LIN {X 0,Y 255.969,Z 835.136,A -85,B 0,C 180,E1 -27165.742,E2 -27165.742} C_VEL
LIN {X 0,Y 253.083,Z 837.367,A -85,B 0,C 180,E1 -27167.208,E2 -27167.208} C_VEL
LIN {X 0,Y 247.96,Z 840.393,A -85,B 0,C 180,E1 -27170.241,E2 -27170.241} C_VEL
LIN {X 0,Y 243.682,Z 841.765,A -85,B 0,C 180,E1 -27173.397,E2 -27173.397} C_VEL
LIN {X 0,Y 241.91,Z 841.979,A -85,B 0,C 180,E1 -27175.016,E2 -27175.016} C_VEL
LIN {X 0,Y 239.218,Z 841.037,A -85,B 0,C 180,E1 -27178.322,E2 -27178.322} C_VEL
LIN {X 0,Y 237.369,Z 838.544,A -85,B 0,C 180,E1 -27181.69,E2 -27181.69} C_VEL
LIN {X 0,Y 236.528,Z 835.644,A -85,B 0,C 180,E1 -27184.245,E2 -27184.245} C_VEL
LIN {X 0,Y 236.07,Z 831.744,A -85,B 0,C 180,E1 -27186.816,E2 -27186.816} C_VEL
LIN {X 0,Y 236.118,Z 826.783,A -85,B 0,C 180,E1 -27189.39,E2 -27189.39} C_VEL
LIN {X 0,Y 236.294,Z 821.698,A -85,B 0,C 180,E1 -27191.551,E2 -27191.551} C_VEL
LIN {X 0,Y 236.654,Z 814.142,A -85,B 0,C 180,E1 -27194.133,E2 -27194.133} C_VEL
LIN {X 0,Y 237.029,Z 806.345,A -85,B 0,C 180,E1 -27196.303,E2 -27196.303} C_VEL
LIN {X 0,Y 237.449,Z 797.897,A -85,B 0,C 180,E1 -27198.265,E2 -27198.265} C_VEL
LIN {X 0,Y 237.963,Z 788.686,A -85,B 0,C 180,E1 -27200.055,E2 -27200.055} C_VEL
LIN {X 0,Y 238.5,Z 779.618,A -85,B 0,C 180,E1 -27201.537,E2 -27201.537} C_VEL
LIN {X 0,Y 239.065,Z 770.085,A -85,B 0,C 180,E1 -27202.843,E2 -27202.843} C_VEL
LIN {X 0,Y 239.688,Z 759.488,A -85,B 0,C 180,E1 -27204.034,E2 -27204.034} C_VEL
LIN {X 0,Y 240.123,Z 749.746,A -85,B 0,C 180,E1 -27204.918,E2 -27204.918} C_VEL
LIN {X 0,Y 240.469,Z 738.64,A -85,B 0,C 180,E1 -27205.698,E2 -27205.698} C_VEL
LIN {X 0,Y 241.686,Z 705.322,A -85,B 0,C 180,E1 -27207.392,E2 -27207.392} C_VEL
LIN {X 0,Y 242.808,Z 665.259,A -85,B 0,C 180,E1 -27209.316,E2 -27209.316} C_VEL
LIN {X 0,Y 240.288,Z 637.438,A -85,B 0,C 180,E1 -27210.679,E2 -27210.679} C_VEL
LIN {X 0,Y 239.995,Z 630.334,A -85,B 0,C 180,E1 -27211.063,E2 -27211.063} C_VEL
LIN {X 0,Y 239.543,Z 627.579,A -85,B 0,C 180,E1 -27212.273,E2 -27212.273} C_VEL
LIN {X 0,Y 239.08,Z 627.634,A -85,B 0,C 180,E1 -27217.969,E2 -27217.969} C_VEL
LIN {X 0,Y 239.069,Z 627.637,A -85,B 0,C 180,E1 -27222.366,E2 -27222.366} C_VEL
LIN {X 0,Y 239.081,Z 627.631,A -85,B 0,C 180,E1 -27225.32,E2 -27225.32} C_VEL
LIN {X 0,Y 239.062,Z 627.639,A -85,B 0,C 180,E1 -27229.864,E2 -27229.864} C_VEL
LIN {X 0,Y 239.028,Z 627.641,A -85,B 0,C 180,E1 -27234.12,E2 -27234.12} C_VEL
LIN {X 0,Y 239.074,Z 627.638,A -85,B 0,C 180,E1 -27238.172,E2 -27238.172} C_VEL
LIN {X 0,Y 239.121,Z 627.632,A -85,B 0,C 180,E1 -27242.051,E2 -27242.051} C_VEL
LIN {X 0,Y 239.152,Z 627.623,A -85,B 0,C 180,E1 -27245.792,E2 -27245.792} C_VEL
LIN {X 0,Y 239.202,Z 627.62,A -85,B 0,C 180,E1 -27249.558,E2 -27249.558} C_VEL
LIN {X 0,Y 239.321,Z 627.599,A -85,B 0,C 180,E1 -27254.978,E2 -27254.978} C_VEL
LIN {X 0,Y 239.388,Z 627.599,A -85,B 0,C 180,E1 -27259.888,E2 -27259.888} C_VEL
LIN {X 0,Y 239.662,Z 627.561,A -85,B 0,C 180,E1 -27263.554,E2 -27263.554} C_VEL
LIN {X 0,Y 239.728,Z 627.552,A -85,B 0,C 180,E1 -27266.65,E2 -27266.65} C_VEL
LIN {X 0,Y 239.869,Z 627.54,A -85,B 0,C 180,E1 -27270,E2 -27270} C_VEL
LIN {X 0,Y 239.728,Z 627.552,A -85,B 0,C 180,E1 -27273.35,E2 -27273.35} C_VEL
LIN {X 0,Y 239.62,Z 627.566,A -85,B 0,C 180,E1 -27276.714,E2 -27276.714} C_VEL
LIN {X 0,Y 239.355,Z 627.603,A -85,B 0,C 180,E1 -27281.82,E2 -27281.82} C_VEL
LIN {X 0,Y 239.296,Z 627.603,A -85,B 0,C 180,E1 -27285.274,E2 -27285.274} C_VEL
LIN {X 0,Y 239.191,Z 627.621,A -85,B 0,C 180,E1 -27290.573,E2 -27290.573} C_VEL
LIN {X 0,Y 239.135,Z 627.623,A -85,B 0,C 180,E1 -27294.77,E2 -27294.77} C_VEL
LIN {X 0,Y 239.118,Z 627.631,A -85,B 0,C 180,E1 -27298.506,E2 -27298.506} C_VEL
LIN {X 0,Y 239.094,Z 627.635,A -85,B 0,C 180,E1 -27301.836,E2 -27301.836} C_VEL
LIN {X 0,Y 239.124,Z 627.628,A -85,B 0,C 180,E1 -27305.862,E2 -27305.862} C_VEL
LIN {X 0,Y 239.097,Z 627.633,A -85,B 0,C 180,E1 -27310.389,E2 -27310.389} C_VEL
LIN {X 0,Y 239.09,Z 627.63,A -85,B 0,C 180,E1 -27314.677,E2 -27314.677} C_VEL
LIN {X 0,Y 239.091,Z 627.634,A -85,B 0,C 180,E1 -27317.639,E2 -27317.639} C_VEL
LIN {X 0,Y 239.091,Z 627.633,A -85,B 0,C 180,E1 -27322.033,E2 -27322.033} C_VEL
LIN {X 0,Y 239.093,Z 627.635,A -85,B 0,C 180,E1 -27326.178,E2 -27326.178} C_VEL
LIN {X 0,Y 239.071,Z 627.637,A -85,B 0,C 180,E1 -27330.128,E2 -27330.128} C_VEL
LIN {X 0,Y 239.107,Z 627.629,A -85,B 0,C 180,E1 -27333.934,E2 -27333.934} C_VEL
LIN {X 0,Y 239.112,Z 627.632,A -85,B 0,C 180,E1 -27337.616,E2 -27337.616} C_VEL
LIN {X 0,Y 239.174,Z 627.621,A -85,B 0,C 180,E1 -27341.208,E2 -27341.208} C_VEL
LIN {X 0,Y 239.271,Z 627.609,A -85,B 0,C 180,E1 -27345.026,E2 -27345.026} C_VEL
LIN {X 0,Y 239.384,Z 627.6,A -85,B 0,C 180,E1 -27349.889,E2 -27349.889} C_VEL
LIN {X 0,Y 239.717,Z 627.551,A -85,B 0,C 180,E1 -27353.446,E2 -27353.446} C_VEL
LIN {X 0,Y 239.736,Z 627.553,A -85,B 0,C 180,E1 -27356.651,E2 -27356.651} C_VEL
LIN {X 0,Y 239.87,Z 627.538,A -85,B 0,C 180,E1 -27360.001,E2 -27360.001} C_VEL
LIN {X 0,Y 239.73,Z 627.549,A -85,B 0,C 180,E1 -27363.351,E2 -27363.351} C_VEL
LIN {X 0,Y 239.623,Z 627.567,A -85,B 0,C 180,E1 -27366.715,E2 -27366.715} C_VEL
LIN {X 0,Y 239.305,Z 627.605,A -85,B 0,C 180,E1 -27371.823,E2 -27371.823} C_VEL
LIN {X 0,Y 239.217,Z 627.617,A -85,B 0,C 180,E1 -27375.28,E2 -27375.28} C_VEL
LIN {X 0,Y 239.138,Z 627.624,A -85,B 0,C 180,E1 -27380.579,E2 -27380.579} C_VEL
LIN {X 0,Y 239.138,Z 627.627,A -85,B 0,C 180,E1 -27384.77,E2 -27384.77} C_VEL
LIN {X 0,Y 239.118,Z 627.63,A -85,B 0,C 180,E1 -27388.504,E2 -27388.504} C_VEL
LIN {X 0,Y 239.076,Z 627.633,A -85,B 0,C 180,E1 -27391.828,E2 -27391.828} C_VEL
LIN {X 0,Y 239.028,Z 627.644,A -85,B 0,C 180,E1 -27395.88,E2 -27395.88} C_VEL
LIN {X 0,Y 239.059,Z 627.635,A -85,B 0,C 180,E1 -27400.136,E2 -27400.136} C_VEL
LIN {X 0,Y 239.041,Z 627.64,A -85,B 0,C 180,E1 -27404.689,E2 -27404.689} C_VEL
LIN {X 0,Y 239.021,Z 627.643,A -85,B 0,C 180,E1 -27407.623,E2 -27407.623} C_VEL
LIN {X 0,Y 239.055,Z 627.636,A -85,B 0,C 180,E1 -27412.026,E2 -27412.026} C_VEL
LIN {X 0,Y 239.072,Z 627.638,A -85,B 0,C 180,E1 -27416.174,E2 -27416.174} C_VEL
LIN {X 0,Y 239.09,Z 627.631,A -85,B 0,C 180,E1 -27420.13,E2 -27420.13} C_VEL
LIN {X 0,Y 239.45,Z 627.719,A -85,B 0,C 180,E1 -27423.565,E2 -27423.565} C_VEL
LIN {X 0,Y 240.611,Z 633.644,A -85,B 0,C 180,E1 -27425.949,E2 -27425.949} C_VEL
LIN {X 0,Y 240.293,Z 637.031,A -85,B 0,C 180,E1 -27427.28,E2 -27427.28} C_VEL
LIN {X 0,Y 239.534,Z 641.423,A -85,B 0,C 180,E1 -27428.963,E2 -27428.963} C_VEL
LIN {X 0,Y 240.199,Z 661.866,A -85,B 0,C 180,E1 -27429.962,E2 -27429.962} C_VEL
LIN {X 0,Y 242.502,Z 689.559,A -85,B 0,C 180,E1 -27431.311,E2 -27431.311} C_VEL
LIN {X 0,Y 240.805,Z 746.631,A -85,B 0,C 180,E1 -27434.117,E2 -27434.117} C_VEL
LIN {X 0,Y 240.33,Z 758.435,A -85,B 0,C 180,E1 -27434.901,E2 -27434.901} C_VEL
LIN {X 0,Y 239.916,Z 769.202,A -85,B 0,C 180,E1 -27435.847,E2 -27435.847} C_VEL
LIN {X 0,Y 239.736,Z 772.319,A -85,B 0,C 180,E1 -27436.16,E2 -27436.16} C_VEL
LIN {X 0,Y 239.264,Z 775.883,A -85,B 0,C 180,E1 -27436.545,E2 -27436.545} C_VEL
LIN {X 0,Y 236.945,Z 782.54,A -85,B 0,C 180,E1 -27437.412,E2 -27437.412} C_VEL
LIN {X 0,Y 232.121,Z 793.434,A -85,B 0,C 180,E1 -27439.214,E2 -27439.214} C_VEL
LIN {X 0,Y 231.246,Z 798.101,A -85,B 0,C 180,E1 -27440.079,E2 -27440.079} C_VEL
LIN {X 0,Y 230.873,Z 806.382,A -85,B 0,C 180,E1 -27441.715,E2 -27441.715} C_VEL
LIN {X 0,Y 230.528,Z 813.892,A -85,B 0,C 180,E1 -27443.458,E2 -27443.458} C_VEL
LIN {X 0,Y 230.407,Z 820.396,A -85,B 0,C 180,E1 -27445.205,E2 -27445.205} C_VEL
LIN {X 0,Y 230.245,Z 827.124,A -85,B 0,C 180,E1 -27447.385,E2 -27447.385} C_VEL
LIN {X 0,Y 230.066,Z 833.651,A -85,B 0,C 180,E1 -27450,E2 -27450} C_VEL
LIN {X 0,Y 229.927,Z 837.306,A -85,B 0,C 180,E1 -27451.746,E2 -27451.746} C_VEL
LIN {X 0,Y 229.564,Z 842.85,A -85,B 0,C 180,E1 -27455.252,E2 -27455.252} C_VEL
LIN {X 0,Y 229.53,Z 844.969,A -85,B 0,C 180,E1 -27457.012,E2 -27457.012} C_VEL
LIN {X 0,Y 230.453,Z 848.056,A -85,B 0,C 180,E1 -27460.508,E2 -27460.508} C_VEL
LIN {X 0,Y 232.38,Z 849.575,A -85,B 0,C 180,E1 -27463.954,E2 -27463.954} C_VEL
LIN {X 0,Y 235.467,Z 849.632,A -85,B 0,C 180,E1 -27467.306,E2 -27467.306} C_VEL
LIN {X 0,Y 237.383,Z 849.211,A -85,B 0,C 180,E1 -27468.94,E2 -27468.94} C_VEL
LIN {X 0,Y 241.904,Z 847.088,A -85,B 0,C 180,E1 -27472.113,E2 -27472.113} C_VEL
LIN {X 0,Y 245.879,Z 844.5,A -85,B 0,C 180,E1 -27474.398,E2 -27474.398} C_VEL
LIN {X 0,Y 252.044,Z 839.532,A -85,B 0,C 180,E1 -27477.294,E2 -27477.294} C_VEL
LIN {X 0,Y 257.146,Z 834.695,A -85,B 0,C 180,E1 -27479.361,E2 -27479.361} C_VEL
LIN {X 0,Y 262.686,Z 828.671,A -85,B 0,C 180,E1 -27481.33,E2 -27481.33} C_VEL
LIN {X 0,Y 268.677,Z 821.348,A -85,B 0,C 180,E1 -27483.194,E2 -27483.194} C_VEL
LIN {X 0,Y 273.992,Z 814.098,A -85,B 0,C 180,E1 -27484.668,E2 -27484.668} C_VEL
LIN {X 0,Y 279.55,Z 805.482,A -85,B 0,C 180,E1 -27486.074,E2 -27486.074} C_VEL
LIN {X 0,Y 284.285,Z 797.291,A -85,B 0,C 180,E1 -27487.132,E2 -27487.132} C_VEL
LIN {X 0,Y 289.766,Z 786.418,A -85,B 0,C 180,E1 -27488.275,E2 -27488.275} C_VEL
LIN {X 0,Y 294.221,Z 776.249,A -85,B 0,C 180,E1 -27489.115,E2 -27489.115} C_VEL
LIN {X 0,Y 298.033,Z 765.844,A -85,B 0,C 180,E1 -27489.825,E2 -27489.825} C_VEL
LIN {X 0,Y 301.383,Z 754.97,A -85,B 0,C 180,E1 -27490.38,E2 -27490.38} C_VEL
LIN {X 0,Y 304.7,Z 740.723,A -85,B 0,C 180,E1 -27490.982,E2 -27490.982} C_VEL
LIN {X 0,Y 306.247,Z 732.083,A -85,B 0,C 180,E1 -27491.312,E2 -27491.312} C_VEL
LIN {X 0,Y 304.844,Z 726.881,A -85,B 0,C 180,E1 -27493.21,E2 -27493.21} C_VEL
LIN {X 0,Y 303.582,Z 722.992,A -85,B 0,C 180,E1 -27495.274,E2 -27495.274} C_VEL
LIN {X 0,Y 302.655,Z 719.169,A -85,B 0,C 180,E1 -27498.363,E2 -27498.363} C_VEL
LIN {X 0,Y 302.452,Z 718.617,A -85,B 0,C 180,E1 -27499.84,E2 -27499.84} C_VEL
LIN {X 0,Y 302.826,Z 718.852,A -85,B 0,C 180,E1 -27502.516,E2 -27502.516} C_VEL
LIN {X 0,Y 304.244,Z 722.091,A -85,B 0,C 180,E1 -27505.819,E2 -27505.819} C_VEL
LIN {X 0,Y 305.607,Z 725.321,A -85,B 0,C 180,E1 -27507.638,E2 -27507.638} C_VEL
LIN {X 0,Y 306.67,Z 728.479,A -85,B 0,C 180,E1 -27508.958,E2 -27508.958} C_VEL
LIN {X 0,Y 302.997,Z 746.766,A -85,B 0,C 180,E1 -27509.657,E2 -27509.657} C_VEL
LIN {X 0,Y 299.281,Z 759.828,A -85,B 0,C 180,E1 -27510.346,E2 -27510.346} C_VEL
LIN {X 0,Y 295.517,Z 770.423,A -85,B 0,C 180,E1 -27511.064,E2 -27511.064} C_VEL
LIN {X 0,Y 291.043,Z 781.07,A -85,B 0,C 180,E1 -27512.011,E2 -27512.011} C_VEL
LIN {X 0,Y 286.235,Z 790.813,A -85,B 0,C 180,E1 -27513.082,E2 -27513.082} C_VEL
LIN {X 0,Y 282.131,Z 798.294,A -85,B 0,C 180,E1 -27514.071,E2 -27514.071} C_VEL
LIN {X 0,Y 277.047,Z 806.464,A -85,B 0,C 180,E1 -27515.39,E2 -27515.39} C_VEL
LIN {X 0,Y 271.848,Z 813.824,A -85,B 0,C 180,E1 -27516.863,E2 -27516.863} C_VEL
LIN {X 0,Y 266.753,Z 820.185,A -85,B 0,C 180,E1 -27518.431,E2 -27518.431} C_VEL
LIN {X 0,Y 261.584,Z 825.975,A -85,B 0,C 180,E1 -27520.187,E2 -27520.187} C_VEL
LIN {X 0,Y 257.596,Z 830.02,A -85,B 0,C 180,E1 -27521.695,E2 -27521.695} C_VEL
LIN {X 0,Y 252.276,Z 834.546,A -85,B 0,C 180,E1 -27523.88,E2 -27523.88} C_VEL
LIN {X 0,Y 246.147,Z 838.668,A -85,B 0,C 180,E1 -27526.841,E2 -27526.841} C_VEL
LIN {X 0,Y 242.87,Z 840.464,A -85,B 0,C 180,E1 -27528.689,E2 -27528.689} C_VEL
LIN {X 0,Y 238.623,Z 841.904,A -85,B 0,C 180,E1 -27531.56,E2 -27531.56} C_VEL
LIN {X 0,Y 234.798,Z 842.001,A -85,B 0,C 180,E1 -27534.865,E2 -27534.865} C_VEL
LIN {X 0,Y 233.286,Z 841.573,A -85,B 0,C 180,E1 -27536.557,E2 -27536.557} C_VEL
LIN {X 0,Y 231.064,Z 839.415,A -85,B 0,C 180,E1 -27539.999,E2 -27539.999} C_VEL
LIN {X 0,Y 229.918,Z 836.807,A -85,B 0,C 180,E1 -27542.619,E2 -27542.619} C_VEL
LIN {X 0,Y 229.245,Z 833.24,A -85,B 0,C 180,E1 -27545.259,E2 -27545.259} C_VEL
LIN {X 0,Y 229.024,Z 828.587,A -85,B 0,C 180,E1 -27547.91,E2 -27547.91} C_VEL
LIN {X 0,Y 229.285,Z 821.172,A -85,B 0,C 180,E1 -27551.175,E2 -27551.175} C_VEL
LIN {X 0,Y 229.589,Z 814.033,A -85,B 0,C 180,E1 -27553.676,E2 -27553.676} C_VEL
LIN {X 0,Y 229.903,Z 808.052,A -85,B 0,C 180,E1 -27555.46,E2 -27555.46} C_VEL
LIN {X 0,Y 230.325,Z 798.974,A -85,B 0,C 180,E1 -27557.704,E2 -27557.704} C_VEL
LIN {X 0,Y 230.833,Z 790.228,A -85,B 0,C 180,E1 -27559.498,E2 -27559.498} C_VEL
LIN {X 0,Y 231.31,Z 781.035,A -85,B 0,C 180,E1 -27561.083,E2 -27561.083} C_VEL
LIN {X 0,Y 231.965,Z 770.074,A -85,B 0,C 180,E1 -27562.643,E2 -27562.643} C_VEL
LIN {X 0,Y 232.541,Z 760.56,A -85,B 0,C 180,E1 -27563.757,E2 -27563.757} C_VEL
LIN {X 0,Y 233.025,Z 749.841,A -85,B 0,C 180,E1 -27564.767,E2 -27564.767} C_VEL
LIN {X 0,Y 233.376,Z 739.04,A -85,B 0,C 180,E1 -27565.553,E2 -27565.553} C_VEL
LIN {X 0,Y 234.237,Z 715.097,A -85,B 0,C 180,E1 -27566.83,E2 -27566.83} C_VEL
LIN {X 0,Y 235.787,Z 666.248,A -85,B 0,C 180,E1 -27569.3,E2 -27569.3} C_VEL
LIN {X 0,Y 233.191,Z 637.147,A -85,B 0,C 180,E1 -27570.768,E2 -27570.768} C_VEL
LIN {X 0,Y 232.898,Z 630.557,A -85,B 0,C 180,E1 -27571.125,E2 -27571.125} C_VEL
LIN {X 0,Y 232.529,Z 628.453,A -85,B 0,C 180,E1 -27572.132,E2 -27572.132} C_VEL
LIN {X 0,Y 232.013,Z 628.516,A -85,B 0,C 180,E1 -27578.285,E2 -27578.285} C_VEL
LIN {X 0,Y 232.009,Z 628.517,A -85,B 0,C 180,E1 -27581.619,E2 -27581.619} C_VEL
LIN {X 0,Y 232.034,Z 628.51,A -85,B 0,C 180,E1 -27586.028,E2 -27586.028} C_VEL
LIN {X 0,Y 231.995,Z 628.518,A -85,B 0,C 180,E1 -27590.651,E2 -27590.651} C_VEL
LIN {X 0,Y 232.012,Z 628.511,A -85,B 0,C 180,E1 -27594.997,E2 -27594.997} C_VEL
LIN {X 0,Y 232.016,Z 628.514,A -85,B 0,C 180,E1 -27599.121,E2 -27599.121} C_VEL
LIN {X 0,Y 232.062,Z 628.508,A -85,B 0,C 180,E1 -27603.079,E2 -27603.079} C_VEL
LIN {X 0,Y 232.082,Z 628.503,A -85,B 0,C 180,E1 -27606.899,E2 -27606.899} C_VEL
LIN {X 0,Y 232.135,Z 628.5,A -85,B 0,C 180,E1 -27610.615,E2 -27610.615} C_VEL
LIN {X 0,Y 232.283,Z 628.479,A -85,B 0,C 180,E1 -27616.04,E2 -27616.04} C_VEL
LIN {X 0,Y 232.402,Z 628.467,A -85,B 0,C 180,E1 -27621.332,E2 -27621.332} C_VEL
LIN {X 0,Y 232.593,Z 628.437,A -85,B 0,C 180,E1 -27624.816,E2 -27624.816} C_VEL
LIN {X 0,Y 232.694,Z 628.432,A -85,B 0,C 180,E1 -27628.275,E2 -27628.275} C_VEL
LIN {X 0,Y 232.835,Z 628.417,A -85,B 0,C 180,E1 -27630,E2 -27630} C_VEL
LIN {X 0,Y 232.696,Z 628.428,A -85,B 0,C 180,E1 -27633.451,E2 -27633.451} C_VEL
LIN {X 0,Y 232.545,Z 628.447,A -85,B 0,C 180,E1 -27636.92,E2 -27636.92} C_VEL
LIN {X 0,Y 232.289,Z 628.481,A -85,B 0,C 180,E1 -27642.185,E2 -27642.185} C_VEL
LIN {X 0,Y 232.199,Z 628.489,A -85,B 0,C 180,E1 -27645.753,E2 -27645.753} C_VEL
LIN {X 0,Y 232.155,Z 628.497,A -85,B 0,C 180,E1 -27650.723,E2 -27650.723} C_VEL
LIN {X 0,Y 232.085,Z 628.501,A -85,B 0,C 180,E1 -27655.123,E2 -27655.123} C_VEL
LIN {X 0,Y 232.057,Z 628.51,A -85,B 0,C 180,E1 -27658.916,E2 -27658.916} C_VEL
LIN {X 0,Y 232.051,Z 628.506,A -85,B 0,C 180,E1 -27662.91,E2 -27662.91} C_VEL
LIN {X 0,Y 232.051,Z 628.509,A -85,B 0,C 180,E1 -27667.135,E2 -27667.135} C_VEL
LIN {X 0,Y 232.029,Z 628.513,A -85,B 0,C 180,E1 -27671.615,E2 -27671.615} C_VEL
LIN {X 0,Y 232.041,Z 628.513,A -85,B 0,C 180,E1 -27676.031,E2 -27676.031} C_VEL
LIN {X 0,Y 232.031,Z 628.512,A -85,B 0,C 180,E1 -27680.66,E2 -27680.66} C_VEL
LIN {X 0,Y 232.055,Z 628.507,A -85,B 0,C 180,E1 -27685.006,E2 -27685.006} C_VEL
LIN {X 0,Y 232.016,Z 628.515,A -85,B 0,C 180,E1 -27689.122,E2 -27689.122} C_VEL
LIN {X 0,Y 232.063,Z 628.503,A -85,B 0,C 180,E1 -27693.08,E2 -27693.08} C_VEL
LIN {X 0,Y 232.072,Z 628.507,A -85,B 0,C 180,E1 -27696.899,E2 -27696.899} C_VEL
LIN {X 0,Y 232.114,Z 628.501,A -85,B 0,C 180,E1 -27700.614,E2 -27700.614} C_VEL
LIN {X 0,Y 232.228,Z 628.486,A -85,B 0,C 180,E1 -27704.835,E2 -27704.835} C_VEL
LIN {X 0,Y 232.308,Z 628.479,A -85,B 0,C 180,E1 -27709.578,E2 -27709.578} C_VEL
LIN {X 0,Y 232.666,Z 628.429,A -85,B 0,C 180,E1 -27713.447,E2 -27713.447} C_VEL
LIN {X 0,Y 232.705,Z 628.43,A -85,B 0,C 180,E1 -27716.549,E2 -27716.549} C_VEL
LIN {X 0,Y 232.835,Z 628.414,A -85,B 0,C 180,E1 -27720.001,E2 -27720.001} C_VEL
LIN {X 0,Y 232.699,Z 628.425,A -85,B 0,C 180,E1 -27723.452,E2 -27723.452} C_VEL
LIN {X 0,Y 232.548,Z 628.448,A -85,B 0,C 180,E1 -27726.92,E2 -27726.92} C_VEL
LIN {X 0,Y 232.235,Z 628.485,A -85,B 0,C 180,E1 -27732.189,E2 -27732.189} C_VEL
LIN {X 0,Y 232.153,Z 628.499,A -85,B 0,C 180,E1 -27735.757,E2 -27735.757} C_VEL
LIN {X 0,Y 232.084,Z 628.502,A -85,B 0,C 180,E1 -27740.675,E2 -27740.675} C_VEL
LIN {X 0,Y 232.088,Z 628.505,A -85,B 0,C 180,E1 -27745.123,E2 -27745.123} C_VEL
LIN {X 0,Y 232.056,Z 628.508,A -85,B 0,C 180,E1 -27748.915,E2 -27748.915} C_VEL
LIN {X 0,Y 232.01,Z 628.512,A -85,B 0,C 180,E1 -27752.918,E2 -27752.918} C_VEL
LIN {X 0,Y 231.995,Z 628.517,A -85,B 0,C 180,E1 -27757.146,E2 -27757.146} C_VEL
LIN {X 0,Y 231.978,Z 628.516,A -85,B 0,C 180,E1 -27761.627,E2 -27761.627} C_VEL
LIN {X 0,Y 231.972,Z 628.524,A -85,B 0,C 180,E1 -27766.014,E2 -27766.014} C_VEL
LIN {X 0,Y 231.993,Z 628.512,A -85,B 0,C 180,E1 -27770.651,E2 -27770.651} C_VEL
LIN {X 0,Y 232.012,Z 628.515,A -85,B 0,C 180,E1 -27774.998,E2 -27774.998} C_VEL
LIN {X 0,Y 232.025,Z 628.511,A -85,B 0,C 180,E1 -27779.123,E2 -27779.123} C_VEL
LIN {X 0,Y 232.431,Z 628.559,A -85,B 0,C 180,E1 -27783.722,E2 -27783.722} C_VEL
LIN {X 0,Y 233.539,Z 634.342,A -85,B 0,C 180,E1 -27786.115,E2 -27786.115} C_VEL
LIN {X 0,Y 232.455,Z 641.113,A -85,B 0,C 180,E1 -27788.858,E2 -27788.858} C_VEL
LIN {X 0,Y 233.082,Z 661.522,A -85,B 0,C 180,E1 -27789.904,E2 -27789.904} C_VEL
LIN {X 0,Y 235.356,Z 690.045,A -85,B 0,C 180,E1 -27791.342,E2 -27791.342} C_VEL
LIN {X 0,Y 233.731,Z 746.504,A -85,B 0,C 180,E1 -27794.246,E2 -27794.246} C_VEL
LIN {X 0,Y 233.288,Z 757.483,A -85,B 0,C 180,E1 -27794.992,E2 -27794.992} C_VEL
LIN {X 0,Y 232.885,Z 768.4,A -85,B 0,C 180,E1 -27795.967,E2 -27795.967} C_VEL
LIN {X 0,Y 232.378,Z 778.933,A -85,B 0,C 180,E1 -27797.156,E2 -27797.156} C_VEL
LIN {X 0,Y 231.772,Z 788.297,A -85,B 0,C 180,E1 -27798.451,E2 -27798.451} C_VEL
LIN {X 0,Y 231.362,Z 796.338,A -85,B 0,C 180,E1 -27799.755,E2 -27799.755} C_VEL
LIN {X 0,Y 231.246,Z 798.101,A -85,B 0,C 180,E1 -27800.079,E2 -27800.079} C_VEL
LIN {X 0,Y 230.404,Z 802.726,A -85,B 0,C 180,E1 -27800.965,E2 -27800.965} C_VEL
LIN {X 0,Y 227.31,Z 809.581,A -85,B 0,C 180,E1 -27802.589,E2 -27802.589} C_VEL
LIN {X 0,Y 224.235,Z 815.899,A -85,B 0,C 180,E1 -27804.391,E2 -27804.391} C_VEL
LIN {X 0,Y 223.469,Z 819.618,A -85,B 0,C 180,E1 -27805.566,E2 -27805.566} C_VEL
LIN {X 0,Y 223.313,Z 827.429,A -85,B 0,C 180,E1 -27808.203,E2 -27808.203} C_VEL
LIN {X 0,Y 223.147,Z 831.936,A -85,B 0,C 180,E1 -27810,E2 -27810} C_VEL
LIN {X 0,Y 222.817,Z 837.406,A -85,B 0,C 180,E1 -27812.703,E2 -27812.703} C_VEL
LIN {X 0,Y 222.587,Z 841.646,A -85,B 0,C 180,E1 -27815.417,E2 -27815.417} C_VEL
LIN {X 0,Y 222.854,Z 845.74,A -85,B 0,C 180,E1 -27819.042,E2 -27819.042} C_VEL
LIN {X 0,Y 224.423,Z 848.328,A -85,B 0,C 180,E1 -27822.62,E2 -27822.62} C_VEL
LIN {X 0,Y 225.504,Z 849.154,A -85,B 0,C 180,E1 -27824.389,E2 -27824.389} C_VEL
LIN {X 0,Y 228.697,Z 849.601,A -85,B 0,C 180,E1 -27827.835,E2 -27827.835} C_VEL
LIN {X 0,Y 233.413,Z 848.295,A -85,B 0,C 180,E1 -27831.522,E2 -27831.522} C_VEL
LIN {X 0,Y 238.017,Z 846.001,A -85,B 0,C 180,E1 -27834.331,E2 -27834.331} C_VEL
LIN {X 0,Y 242.556,Z 843.137,A -85,B 0,C 180,E1 -27836.59,E2 -27836.59} C_VEL
LIN {X 0,Y 247.543,Z 839.324,A -85,B 0,C 180,E1 -27838.753,E2 -27838.753} C_VEL
LIN {X 0,Y 252.95,Z 834.469,A -85,B 0,C 180,E1 -27840.816,E2 -27840.816} C_VEL
LIN {X 0,Y 259.515,Z 827.752,A -85,B 0,C 180,E1 -27842.993,E2 -27842.993} C_VEL
LIN {X 0,Y 265.128,Z 821.259,A -85,B 0,C 180,E1 -27844.612,E2 -27844.612} C_VEL
LIN {X 0,Y 270.652,Z 814.001,A -85,B 0,C 180,E1 -27846.07,E2 -27846.07} C_VEL
LIN {X 0,Y 276.447,Z 805.455,A -85,B 0,C 180,E1 -27847.452,E2 -27847.452} C_VEL
LIN {X 0,Y 281.999,Z 796.304,A -85,B 0,C 180,E1 -27848.614,E2 -27848.614} C_VEL
LIN {X 0,Y 286.434,Z 787.977,A -85,B 0,C 180,E1 -27849.48,E2 -27849.48} C_VEL
LIN {X 0,Y 290.998,Z 778.115,A -85,B 0,C 180,E1 -27850.308,E2 -27850.308} C_VEL
LIN {X 0,Y 294.944,Z 768.048,A -85,B 0,C 180,E1 -27851,E2 -27851} C_VEL
LIN {X 0,Y 298.418,Z 757.549,A -85,B 0,C 180,E1 -27851.566,E2 -27851.566} C_VEL
LIN {X 0,Y 301.567,Z 745.744,A -85,B 0,C 180,E1 -27852.078,E2 -27852.078} C_VEL
LIN {X 0,Y 303.56,Z 736.488,A -85,B 0,C 180,E1 -27852.415,E2 -27852.415} C_VEL
LIN {X 0,Y 302.477,Z 732.456,A -85,B 0,C 180,E1 -27854.056,E2 -27854.056} C_VEL
LIN {X 0,Y 301.739,Z 729.655,A -85,B 0,C 180,E1 -27855.586,E2 -27855.586} C_VEL
LIN {X 0,Y 300.957,Z 725.89,A -85,B 0,C 180,E1 -27858.725,E2 -27858.725} C_VEL
LIN {X 0,Y 300.891,Z 725.466,A -85,B 0,C 180,E1 -27861.058,E2 -27861.058} C_VEL
LIN {X 0,Y 301.183,Z 725.905,A -85,B 0,C 180,E1 -27862.621,E2 -27862.621} C_VEL
LIN {X 0,Y 302.366,Z 728.664,A -85,B 0,C 180,E1 -27865.454,E2 -27865.454} C_VEL
LIN {X 0,Y 303.657,Z 732.07,A -85,B 0,C 180,E1 -27867.388,E2 -27867.388} C_VEL
LIN {X 0,Y 303.935,Z 733.24,A -85,B 0,C 180,E1 -27867.828,E2 -27867.828} C_VEL
LIN {X 0,Y 300.28,Z 749.351,A -85,B 0,C 180,E1 -27868.471,E2 -27868.471} C_VEL
LIN {X 0,Y 296.74,Z 760.842,A -85,B 0,C 180,E1 -27869.09,E2 -27869.09} C_VEL
LIN {X 0,Y 292.661,Z 771.806,A -85,B 0,C 180,E1 -27869.827,E2 -27869.827} C_VEL
LIN {X 0,Y 288.946,Z 780.454,A -85,B 0,C 180,E1 -27870.58,E2 -27870.58} C_VEL
LIN {X 0,Y 284.491,Z 789.373,A -85,B 0,C 180,E1 -27871.508,E2 -27871.508} C_VEL
LIN {X 0,Y 279.02,Z 798.817,A -85,B 0,C 180,E1 -27872.732,E2 -27872.732} C_VEL
LIN {X 0,Y 273.188,Z 807.575,A -85,B 0,C 180,E1 -27874.159,E2 -27874.159} C_VEL
LIN {X 0,Y 268.737,Z 813.647,A -85,B 0,C 180,E1 -27875.352,E2 -27875.352} C_VEL
LIN {X 0,Y 263.423,Z 820.093,A -85,B 0,C 180,E1 -27876.908,E2 -27876.908} C_VEL
LIN {X 0,Y 258.305,Z 825.553,A -85,B 0,C 180,E1 -27878.526,E2 -27878.526} C_VEL
LIN {X 0,Y 252.551,Z 830.875,A -85,B 0,C 180,E1 -27880.56,E2 -27880.56} C_VEL
LIN {X 0,Y 247.151,Z 835.151,A -85,B 0,C 180,E1 -27882.687,E2 -27882.687} C_VEL
LIN {X 0,Y 242.218,Z 838.376,A -85,B 0,C 180,E1 -27884.914,E2 -27884.914} C_VEL
LIN {X 0,Y 236.205,Z 841.137,A -85,B 0,C 180,E1 -27888.123,E2 -27888.123} C_VEL
LIN {X 0,Y 233.853,Z 841.951,A -85,B 0,C 180,E1 -27889.646,E2 -27889.646} C_VEL
LIN {X 0,Y 229.438,Z 842.373,A -85,B 0,C 180,E1 -27892.985,E2 -27892.985} C_VEL
LIN {X 0,Y 226.149,Z 841.219,A -85,B 0,C 180,E1 -27896.448,E2 -27896.448} C_VEL
LIN {X 0,Y 224.953,Z 840.165,A -85,B 0,C 180,E1 -27898.215,E2 -27898.215} C_VEL
LIN {X 0,Y 223.122,Z 836.757,A -85,B 0,C 180,E1 -27901.798,E2 -27901.798} C_VEL
LIN {X 0,Y 222.377,Z 833.152,A -85,B 0,C 180,E1 -27904.516,E2 -27904.516} C_VEL
LIN {X 0,Y 222.061,Z 828.519,A -85,B 0,C 180,E1 -27907.248,E2 -27907.248} C_VEL
LIN {X 0,Y 222.25,Z 821.51,A -85,B 0,C 180,E1 -27910.44,E2 -27910.44} C_VEL
LIN {X 0,Y 222.478,Z 815.317,A -85,B 0,C 180,E1 -27912.731,E2 -27912.731} C_VEL
LIN {X 0,Y 222.892,Z 807.881,A -85,B 0,C 180,E1 -27915.025,E2 -27915.025} C_VEL
LIN {X 0,Y 223.291,Z 798.77,A -85,B 0,C 180,E1 -27917.337,E2 -27917.337} C_VEL
LIN {X 0,Y 223.785,Z 790.088,A -85,B 0,C 180,E1 -27919.186,E2 -27919.186} C_VEL
LIN {X 0,Y 224.235,Z 781.014,A -85,B 0,C 180,E1 -27920.811,E2 -27920.811} C_VEL
LIN {X 0,Y 224.774,Z 771.838,A -85,B 0,C 180,E1 -27922.199,E2 -27922.199} C_VEL
LIN {X 0,Y 225.389,Z 761.622,A -85,B 0,C 180,E1 -27923.463,E2 -27923.463} C_VEL
LIN {X 0,Y 225.952,Z 749.838,A -85,B 0,C 180,E1 -27924.617,E2 -27924.617} C_VEL
LIN {X 0,Y 226.309,Z 738.949,A -85,B 0,C 180,E1 -27925.431,E2 -27925.431} C_VEL
LIN {X 0,Y 227.538,Z 704.664,A -85,B 0,C 180,E1 -27927.3,E2 -27927.3} C_VEL
LIN {X 0,Y 228.658,Z 666.149,A -85,B 0,C 180,E1 -27929.309,E2 -27929.309} C_VEL
LIN {X 0,Y 226.114,Z 638.202,A -85,B 0,C 180,E1 -27930.776,E2 -27930.776} C_VEL
LIN {X 0,Y 225.811,Z 630.786,A -85,B 0,C 180,E1 -27931.17,E2 -27931.17} C_VEL
LIN {X 0,Y 225.533,Z 629.326,A -85,B 0,C 180,E1 -27931.868,E2 -27931.868} C_VEL
LIN {X 0,Y 225.022,Z 629.382,A -85,B 0,C 180,E1 -27936.257,E2 -27936.257} C_VEL
LIN {X 0,Y 224.978,Z 629.391,A -85,B 0,C 180,E1 -27940.829,E2 -27940.829} C_VEL
LIN {X 0,Y 224.994,Z 629.387,A -85,B 0,C 180,E1 -27945.726,E2 -27945.726} C_VEL
LIN {X 0,Y 224.969,Z 629.391,A -85,B 0,C 180,E1 -27949.168,E2 -27949.168} C_VEL
LIN {X 0,Y 224.952,Z 629.394,A -85,B 0,C 180,E1 -27954.053,E2 -27954.053} C_VEL
LIN {X 0,Y 224.961,Z 629.394,A -85,B 0,C 180,E1 -27958.04,E2 -27958.04} C_VEL
LIN {X 0,Y 225.004,Z 629.39,A -85,B 0,C 180,E1 -27962.163,E2 -27962.163} C_VEL
LIN {X 0,Y 225.005,Z 629.386,A -85,B 0,C 180,E1 -27966.128,E2 -27966.128} C_VEL
LIN {X 0,Y 225.098,Z 629.38,A -85,B 0,C 180,E1 -27969.983,E2 -27969.983} C_VEL
LIN {X 0,Y 225.24,Z 629.355,A -85,B 0,C 180,E1 -27975.594,E2 -27975.594} C_VEL
LIN {X 0,Y 225.35,Z 629.345,A -85,B 0,C 180,E1 -27981.059,E2 -27981.059} C_VEL
LIN {X 0,Y 225.589,Z 629.314,A -85,B 0,C 180,E1 -27983.499,E2 -27983.499} C_VEL
LIN {X 0,Y 225.665,Z 629.305,A -85,B 0,C 180,E1 -27986.441,E2 -27986.441} C_VEL
LIN {X 0,Y 225.786,Z 629.295,A -85,B 0,C 180,E1 -27990,E2 -27990} C_VEL
LIN {X 0,Y 225.664,Z 629.305,A -85,B 0,C 180,E1 -27993.559,E2 -27993.559} C_VEL
LIN {X 0,Y 225.486,Z 629.326,A -85,B 0,C 180,E1 -27997.137,E2 -27997.137} C_VEL
LIN {X 0,Y 225.223,Z 629.359,A -85,B 0,C 180,E1 -28002.574,E2 -28002.574} C_VEL
LIN {X 0,Y 225.11,Z 629.376,A -85,B 0,C 180,E1 -28006.262,E2 -28006.262} C_VEL
LIN {X 0,Y 225.087,Z 629.377,A -85,B 0,C 180,E1 -28011.005,E2 -28011.005} C_VEL
LIN {X 0,Y 225.024,Z 629.384,A -85,B 0,C 180,E1 -28015.835,E2 -28015.835} C_VEL
LIN {X 0,Y 224.985,Z 629.394,A -85,B 0,C 180,E1 -28019.876,E2 -28019.876} C_VEL
LIN {X 0,Y 224.982,Z 629.388,A -85,B 0,C 180,E1 -28024.083,E2 -28024.083} C_VEL
LIN {X 0,Y 225.015,Z 629.388,A -85,B 0,C 180,E1 -28026.259,E2 -28026.259} C_VEL
LIN {X 0,Y 224.998,Z 629.388,A -85,B 0,C 180,E1 -28030.825,E2 -28030.825} C_VEL
LIN {X 0,Y 225.001,Z 629.387,A -85,B 0,C 180,E1 -28035.725,E2 -28035.725} C_VEL
LIN {X 0,Y 224.998,Z 629.389,A -85,B 0,C 180,E1 -28039.176,E2 -28039.176} C_VEL
LIN {X 0,Y 224.983,Z 629.388,A -85,B 0,C 180,E1 -28044.043,E2 -28044.043} C_VEL
LIN {X 0,Y 224.963,Z 629.397,A -85,B 0,C 180,E1 -28048.042,E2 -28048.042} C_VEL
LIN {X 0,Y 225.004,Z 629.385,A -85,B 0,C 180,E1 -28052.164,E2 -28052.164} C_VEL
LIN {X 0,Y 225,Z 629.391,A -85,B 0,C 180,E1 -28056.128,E2 -28056.128} C_VEL
LIN {X 0,Y 225.063,Z 629.383,A -85,B 0,C 180,E1 -28059.981,E2 -28059.981} C_VEL
LIN {X 0,Y 225.201,Z 629.363,A -85,B 0,C 180,E1 -28065.593,E2 -28065.593} C_VEL
LIN {X 0,Y 225.348,Z 629.342,A -85,B 0,C 180,E1 -28071.06,E2 -28071.06} C_VEL
LIN {X 0,Y 225.628,Z 629.305,A -85,B 0,C 180,E1 -28073.42,E2 -28073.42} C_VEL
LIN {X 0,Y 225.674,Z 629.306,A -85,B 0,C 180,E1 -28076.442,E2 -28076.442} C_VEL
LIN {X 0,Y 225.786,Z 629.292,A -85,B 0,C 180,E1 -28080.001,E2 -28080.001} C_VEL
LIN {X 0,Y 225.667,Z 629.302,A -85,B 0,C 180,E1 -28083.56,E2 -28083.56} C_VEL
LIN {X 0,Y 225.489,Z 629.328,A -85,B 0,C 180,E1 -28087.138,E2 -28087.138} C_VEL
LIN {X 0,Y 225.168,Z 629.364,A -85,B 0,C 180,E1 -28092.578,E2 -28092.578} C_VEL
LIN {X 0,Y 225.076,Z 629.381,A -85,B 0,C 180,E1 -28096.266,E2 -28096.266} C_VEL
LIN {X 0,Y 225.039,Z 629.379,A -85,B 0,C 180,E1 -28100.971,E2 -28100.971} C_VEL
LIN {X 0,Y 225.028,Z 629.387,A -85,B 0,C 180,E1 -28105.835,E2 -28105.835} C_VEL
LIN {X 0,Y 224.978,Z 629.392,A -85,B 0,C 180,E1 -28109.878,E2 -28109.878} C_VEL
LIN {X 0,Y 224.937,Z 629.398,A -85,B 0,C 180,E1 -28114.092,E2 -28114.092} C_VEL
LIN {X 0,Y 224.955,Z 629.393,A -85,B 0,C 180,E1 -28118.884,E2 -28118.884} C_VEL
LIN {X 0,Y 224.908,Z 629.397,A -85,B 0,C 180,E1 -28123.249,E2 -28123.249} C_VEL
LIN {X 0,Y 224.908,Z 629.4,A -85,B 0,C 180,E1 -28126.752,E2 -28126.752} C_VEL
LIN {X 0,Y 224.955,Z 629.388,A -85,B 0,C 180,E1 -28131.117,E2 -28131.117} C_VEL
LIN {X 0,Y 224.937,Z 629.4,A -85,B 0,C 180,E1 -28135.909,E2 -28135.909} C_VEL
LIN {X 0,Y 225.022,Z 629.38,A -85,B 0,C 180,E1 -28140.643,E2 -28140.643} C_VEL
LIN {X 0,Y 225.414,Z 629.356,A -85,B 0,C 180,E1 -28143.879,E2 -28143.879} C_VEL
LIN {X 0,Y 226.412,Z 634.99,A -85,B 0,C 180,E1 -28146.286,E2 -28146.286} C_VEL
LIN {X 0,Y 225.361,Z 641.183,A -85,B 0,C 180,E1 -28148.818,E2 -28148.818} C_VEL
LIN {X 0,Y 226.031,Z 662.335,A -85,B 0,C 180,E1 -28149.935,E2 -28149.935} C_VEL
LIN {X 0,Y 228.28,Z 690.034,A -85,B 0,C 180,E1 -28151.38,E2 -28151.38} C_VEL
LIN {X 0,Y 226.669,Z 746.153,A -85,B 0,C 180,E1 -28154.37,E2 -28154.37} C_VEL
LIN {X 0,Y 226.225,Z 757.887,A -85,B 0,C 180,E1 -28155.201,E2 -28155.201} C_VEL
LIN {X 0,Y 225.776,Z 768.612,A -85,B 0,C 180,E1 -28156.203,E2 -28156.203} C_VEL
LIN {X 0,Y 225.308,Z 779.08,A -85,B 0,C 180,E1 -28157.431,E2 -28157.431} C_VEL
LIN {X 0,Y 224.705,Z 788.377,A -85,B 0,C 180,E1 -28158.766,E2 -28158.766} C_VEL
LIN {X 0,Y 224.295,Z 796.361,A -85,B 0,C 180,E1 -28160.11,E2 -28160.11} C_VEL
LIN {X 0,Y 223.909,Z 805.294,A -85,B 0,C 180,E1 -28161.908,E2 -28161.908} C_VEL
LIN {X 0,Y 223.584,Z 812.861,A -85,B 0,C 180,E1 -28163.705,E2 -28163.705} C_VEL
LIN {X 0,Y 223.469,Z 819.618,A -85,B 0,C 180,E1 -28165.566,E2 -28165.566} C_VEL
LIN {X 0,Y 222.74,Z 823.187,A -85,B 0,C 180,E1 -28166.776,E2 -28166.776} C_VEL
LIN {X 0,Y 220.489,Z 827.277,A -85,B 0,C 180,E1 -28168.439,E2 -28168.439} C_VEL
LIN {X 0,Y 217.332,Z 831.816,A -85,B 0,C 180,E1 -28170.635,E2 -28170.635} C_VEL
LIN {X 0,Y 216,Z 835.162,A -85,B 0,C 180,E1 -28172.502,E2 -28172.502} C_VEL
LIN {X 0,Y 215.741,Z 838.805,A -85,B 0,C 180,E1 -28174.656,E2 -28174.656} C_VEL
LIN {X 0,Y 215.631,Z 842.629,A -85,B 0,C 180,E1 -28177.466,E2 -28177.466} C_VEL
LIN {X 0,Y 215.925,Z 844.717,A -85,B 0,C 180,E1 -28179.335,E2 -28179.335} C_VEL
LIN {X 0,Y 217.523,Z 847.701,A -85,B 0,C 180,E1 -28183.027,E2 -28183.027} C_VEL
LIN {X 0,Y 220.238,Z 849.141,A -85,B 0,C 180,E1 -28186.633,E2 -28186.633} C_VEL
LIN {X 0,Y 221.95,Z 849.343,A -85,B 0,C 180,E1 -28188.397,E2 -28188.397} C_VEL
LIN {X 0,Y 226.286,Z 848.743,A -85,B 0,C 180,E1 -28191.805,E2 -28191.805} C_VEL
LIN {X 0,Y 231.593,Z 846.642,A -85,B 0,C 180,E1 -28195.051,E2 -28195.051} C_VEL
LIN {X 0,Y 236.276,Z 844.079,A -85,B 0,C 180,E1 -28197.355,E2 -28197.355} C_VEL
LIN {X 0,Y 243.408,Z 839.012,A -85,B 0,C 180,E1 -28200.334,E2 -28200.334} C_VEL
LIN {X 0,Y 248.974,Z 834.4,A -85,B 0,C 180,E1 -28202.313,E2 -28202.313} C_VEL
LIN {X 0,Y 255.137,Z 828.476,A -85,B 0,C 180,E1 -28204.25,E2 -28204.25} C_VEL
LIN {X 0,Y 261.752,Z 821.201,A -85,B 0,C 180,E1 -28206.066,E2 -28206.066} C_VEL
LIN {X 0,Y 267.534,Z 814.094,A -85,B 0,C 180,E1 -28207.497,E2 -28207.497} C_VEL
LIN {X 0,Y 273.589,Z 805.627,A -85,B 0,C 180,E1 -28208.848,E2 -28208.848} C_VEL
LIN {X 0,Y 279.287,Z 796.527,A -85,B 0,C 180,E1 -28209.991,E2 -28209.991} C_VEL
LIN {X 0,Y 284.527,Z 786.926,A -85,B 0,C 180,E1 -28210.954,E2 -28210.954} C_VEL
LIN {X 0,Y 289.26,Z 777.066,A -85,B 0,C 180,E1 -28211.753,E2 -28211.753} C_VEL
LIN {X 0,Y 293.361,Z 766.977,A -85,B 0,C 180,E1 -28212.417,E2 -28212.417} C_VEL
LIN {X 0,Y 296.753,Z 757.117,A -85,B 0,C 180,E1 -28212.914,E2 -28212.914} C_VEL
LIN {X 0,Y 299.927,Z 745.389,A -85,B 0,C 180,E1 -28213.417,E2 -28213.417} C_VEL
LIN {X 0,Y 300.956,Z 740.927,A -85,B 0,C 180,E1 -28213.598,E2 -28213.598} C_VEL
LIN {X 0,Y 300.342,Z 738.377,A -85,B 0,C 180,E1 -28214.75,E2 -28214.75} C_VEL
LIN {X 0,Y 299.814,Z 735.975,A -85,B 0,C 180,E1 -28216.137,E2 -28216.137} C_VEL
LIN {X 0,Y 299.291,Z 732.755,A -85,B 0,C 180,E1 -28218.864,E2 -28218.864} C_VEL
LIN {X 0,Y 299.205,Z 732.371,A -85,B 0,C 180,E1 -28220.796,E2 -28220.796} C_VEL
LIN {X 0,Y 299.517,Z 732.816,A -85,B 0,C 180,E1 -28222.552,E2 -28222.552} C_VEL
LIN {X 0,Y 300.534,Z 735.403,A -85,B 0,C 180,E1 -28225.186,E2 -28225.186} C_VEL
LIN {X 0,Y 301.376,Z 737.915,A -85,B 0,C 180,E1 -28226.68,E2 -28226.68} C_VEL
LIN {X 0,Y 298.426,Z 749.925,A -85,B 0,C 180,E1 -28227.161,E2 -28227.161} C_VEL
LIN {X 0,Y 294.842,Z 761.216,A -85,B 0,C 180,E1 -28227.745,E2 -28227.745} C_VEL
LIN {X 0,Y 290.886,Z 771.418,A -85,B 0,C 180,E1 -28228.414,E2 -28228.414} C_VEL
LIN {X 0,Y 286.909,Z 780.251,A -85,B 0,C 180,E1 -28229.157,E2 -28229.157} C_VEL
LIN {X 0,Y 281.067,Z 791.288,A -85,B 0,C 180,E1 -28230.31,E2 -28230.31} C_VEL
LIN {X 0,Y 276.682,Z 798.621,A -85,B 0,C 180,E1 -28231.249,E2 -28231.249} C_VEL
LIN {X 0,Y 271.822,Z 805.862,A -85,B 0,C 180,E1 -28232.365,E2 -28232.365} C_VEL
LIN {X 0,Y 265.537,Z 813.933,A -85,B 0,C 180,E1 -28233.893,E2 -28233.893} C_VEL
LIN {X 0,Y 259.191,Z 821.128,A -85,B 0,C 180,E1 -28235.662,E2 -28235.662} C_VEL
LIN {X 0,Y 253.853,Z 826.47,A -85,B 0,C 180,E1 -28237.275,E2 -28237.275} C_VEL
LIN {X 0,Y 248.446,Z 831.187,A -85,B 0,C 180,E1 -28239.08,E2 -28239.08} C_VEL
LIN {X 0,Y 242.122,Z 835.753,A -85,B 0,C 180,E1 -28241.444,E2 -28241.444} C_VEL
LIN {X 0,Y 238.631,Z 837.961,A -85,B 0,C 180,E1 -28242.93,E2 -28242.93} C_VEL
LIN {X 0,Y 232.247,Z 841.033,A -85,B 0,C 180,E1 -28246.038,E2 -28246.038} C_VEL
LIN {X 0,Y 226.797,Z 842.418,A -85,B 0,C 180,E1 -28249.321,E2 -28249.321} C_VEL
LIN {X 0,Y 224.45,Z 842.633,A -85,B 0,C 180,E1 -28251.023,E2 -28251.023} C_VEL
LIN {X 0,Y 220.54,Z 841.802,A -85,B 0,C 180,E1 -28254.532,E2 -28254.532} C_VEL
LIN {X 0,Y 217.843,Z 839.421,A -85,B 0,C 180,E1 -28258.157,E2 -28258.157} C_VEL
LIN {X 0,Y 216.377,Z 836.695,A -85,B 0,C 180,E1 -28260.927,E2 -28260.927} C_VEL
LIN {X 0,Y 215.514,Z 833.018,A -85,B 0,C 180,E1 -28263.726,E2 -28263.726} C_VEL
LIN {X 0,Y 215.102,Z 828.312,A -85,B 0,C 180,E1 -28266.544,E2 -28266.544} C_VEL
LIN {X 0,Y 215.265,Z 821.331,A -85,B 0,C 180,E1 -28269.835,E2 -28269.835} C_VEL
LIN {X 0,Y 215.489,Z 814.777,A -85,B 0,C 180,E1 -28272.327,E2 -28272.327} C_VEL
LIN {X 0,Y 215.891,Z 807.707,A -85,B 0,C 180,E1 -28274.562,E2 -28274.562} C_VEL
LIN {X 0,Y 216.277,Z 798.557,A -85,B 0,C 180,E1 -28276.946,E2 -28276.946} C_VEL
LIN {X 0,Y 216.692,Z 791.034,A -85,B 0,C 180,E1 -28278.614,E2 -28278.614} C_VEL
LIN {X 0,Y 217.154,Z 781.507,A -85,B 0,C 180,E1 -28280.393,E2 -28280.393} C_VEL
LIN {X 0,Y 217.741,Z 771.451,A -85,B 0,C 180,E1 -28281.959,E2 -28281.959} C_VEL
LIN {X 0,Y 218.337,Z 761.259,A -85,B 0,C 180,E1 -28283.265,E2 -28283.265} C_VEL
LIN {X 0,Y 218.819,Z 750.874,A -85,B 0,C 180,E1 -28284.338,E2 -28284.338} C_VEL
LIN {X 0,Y 219.206,Z 739.608,A -85,B 0,C 180,E1 -28285.237,E2 -28285.237} C_VEL
LIN {X 0,Y 220.101,Z 713.982,A -85,B 0,C 180,E1 -28286.724,E2 -28286.724} C_VEL
LIN {X 0,Y 221.514,Z 666.098,A -85,B 0,C 180,E1 -28289.315,E2 -28289.315} C_VEL
LIN {X 0,Y 219.026,Z 637.87,A -85,B 0,C 180,E1 -28290.842,E2 -28290.842} C_VEL
LIN {X 0,Y 218.728,Z 630.964,A -85,B 0,C 180,E1 -28291.223,E2 -28291.223} C_VEL
LIN {X 0,Y 218.56,Z 630.195,A -85,B 0,C 180,E1 -28291.653,E2 -28291.653} C_VEL
LIN {X 0,Y 217.908,Z 630.268,A -85,B 0,C 180,E1 -28297.642,E2 -28297.642} C_VEL
LIN {X 0,Y 217.914,Z 630.272,A -85,B 0,C 180,E1 -28302.328,E2 -28302.328} C_VEL
LIN {X 0,Y 217.954,Z 630.262,A -85,B 0,C 180,E1 -28305.006,E2 -28305.006} C_VEL
LIN {X 0,Y 217.911,Z 630.275,A -85,B 0,C 180,E1 -28309.993,E2 -28309.993} C_VEL
LIN {X 0,Y 217.889,Z 630.271,A -85,B 0,C 180,E1 -28314.644,E2 -28314.644} C_VEL
LIN {X 0,Y 217.911,Z 630.271,A -85,B 0,C 180,E1 -28319.049,E2 -28319.049} C_VEL
LIN {X 0,Y 217.997,Z 630.259,A -85,B 0,C 180,E1 -28324.112,E2 -28324.112} C_VEL
LIN {X 0,Y 218.06,Z 630.253,A -85,B 0,C 180,E1 -28329.308,E2 -28329.308} C_VEL
LIN {X 0,Y 218.177,Z 630.233,A -85,B 0,C 180,E1 -28335.117,E2 -28335.117} C_VEL
LIN {X 0,Y 218.293,Z 630.224,A -85,B 0,C 180,E1 -28340.767,E2 -28340.767} C_VEL
LIN {X 0,Y 218.557,Z 630.19,A -85,B 0,C 180,E1 -28343.458,E2 -28343.458} C_VEL
LIN {X 0,Y 218.623,Z 630.186,A -85,B 0,C 180,E1 -28348.164,E2 -28348.164} C_VEL
LIN {X 0,Y 218.739,Z 630.172,A -85,B 0,C 180,E1 -28350,E2 -28350} C_VEL
LIN {X 0,Y 218.611,Z 630.184,A -85,B 0,C 180,E1 -28353.674,E2 -28353.674} C_VEL
LIN {X 0,Y 218.429,Z 630.206,A -85,B 0,C 180,E1 -28357.369,E2 -28357.369} C_VEL
LIN {X 0,Y 218.162,Z 630.237,A -85,B 0,C 180,E1 -28362.988,E2 -28362.988} C_VEL
LIN {X 0,Y 218.04,Z 630.254,A -85,B 0,C 180,E1 -28366.805,E2 -28366.805} C_VEL
LIN {X 0,Y 218.014,Z 630.259,A -85,B 0,C 180,E1 -28371.298,E2 -28371.298} C_VEL
LIN {X 0,Y 217.996,Z 630.259,A -85,B 0,C 180,E1 -28375.888,E2 -28375.888} C_VEL
LIN {X 0,Y 217.929,Z 630.269,A -85,B 0,C 180,E1 -28380.947,E2 -28380.947} C_VEL
LIN {X 0,Y 217.944,Z 630.264,A -85,B 0,C 180,E1 -28385.345,E2 -28385.345} C_VEL
LIN {X 0,Y 217.936,Z 630.271,A -85,B 0,C 180,E1 -28390,E2 -28390} C_VEL
LIN {X 0,Y 217.952,Z 630.263,A -85,B 0,C 180,E1 -28395.008,E2 -28395.008} C_VEL
LIN {X 0,Y 217.934,Z 630.271,A -85,B 0,C 180,E1 -28400,E2 -28400} C_VEL
LIN {X 0,Y 217.915,Z 630.268,A -85,B 0,C 180,E1 -28404.651,E2 -28404.651} C_VEL
LIN {X 0,Y 217.912,Z 630.271,A -85,B 0,C 180,E1 -28409.051,E2 -28409.051} C_VEL
LIN {X 0,Y 218.003,Z 630.258,A -85,B 0,C 180,E1 -28414.11,E2 -28414.11} C_VEL
LIN {X 0,Y 218.025,Z 630.258,A -85,B 0,C 180,E1 -28419.306,E2 -28419.306} C_VEL
LIN {X 0,Y 218.144,Z 630.24,A -85,B 0,C 180,E1 -28425.116,E2 -28425.116} C_VEL
LIN {X 0,Y 218.287,Z 630.222,A -85,B 0,C 180,E1 -28430.768,E2 -28430.768} C_VEL
LIN {X 0,Y 218.574,Z 630.184,A -85,B 0,C 180,E1 -28433.425,E2 -28433.425} C_VEL
LIN {X 0,Y 218.627,Z 630.185,A -85,B 0,C 180,E1 -28438.165,E2 -28438.165} C_VEL
LIN {X 0,Y 218.739,Z 630.169,A -85,B 0,C 180,E1 -28440.001,E2 -28440.001} C_VEL
LIN {X 0,Y 218.613,Z 630.181,A -85,B 0,C 180,E1 -28443.675,E2 -28443.675} C_VEL
LIN {X 0,Y 218.431,Z 630.208,A -85,B 0,C 180,E1 -28447.37,E2 -28447.37} C_VEL
LIN {X 0,Y 218.182,Z 630.234,A -85,B 0,C 180,E1 -28451.106,E2 -28451.106} C_VEL
LIN {X 0,Y 218.075,Z 630.251,A -85,B 0,C 180,E1 -28455.511,E2 -28455.511} C_VEL
LIN {X 0,Y 218.007,Z 630.255,A -85,B 0,C 180,E1 -28460.697,E2 -28460.697} C_VEL
LIN {X 0,Y 218,Z 630.263,A -85,B 0,C 180,E1 -28465.888,E2 -28465.888} C_VEL
LIN {X 0,Y 217.913,Z 630.266,A -85,B 0,C 180,E1 -28470.951,E2 -28470.951} C_VEL
LIN {X 0,Y 217.889,Z 630.274,A -85,B 0,C 180,E1 -28475.356,E2 -28475.356} C_VEL
LIN {X 0,Y 217.906,Z 630.27,A -85,B 0,C 180,E1 -28480.008,E2 -28480.008} C_VEL
LIN {X 0,Y 217.879,Z 630.275,A -85,B 0,C 180,E1 -28485.013,E2 -28485.013} C_VEL
LIN {X 0,Y 217.906,Z 630.27,A -85,B 0,C 180,E1 -28489.993,E2 -28489.993} C_VEL
LIN {X 0,Y 217.874,Z 630.277,A -85,B 0,C 180,E1 -28494.642,E2 -28494.642} C_VEL
LIN {X 0,Y 217.921,Z 630.268,A -85,B 0,C 180,E1 -28499.051,E2 -28499.051} C_VEL
LIN {X 0,Y 218.462,Z 630.296,A -85,B 0,C 180,E1 -28504.142,E2 -28504.142} C_VEL
LIN {X 0,Y 219.281,Z 634.451,A -85,B 0,C 180,E1 -28505.967,E2 -28505.967} C_VEL
LIN {X 0,Y 218.278,Z 640.888,A -85,B 0,C 180,E1 -28508.757,E2 -28508.757} C_VEL
LIN {X 0,Y 218.931,Z 662.605,A -85,B 0,C 180,E1 -28509.945,E2 -28509.945} C_VEL
LIN {X 0,Y 221.185,Z 691.111,A -85,B 0,C 180,E1 -28511.478,E2 -28511.478} C_VEL
LIN {X 0,Y 219.567,Z 746.711,A -85,B 0,C 180,E1 -28514.564,E2 -28514.564} C_VEL
LIN {X 0,Y 219.148,Z 758.227,A -85,B 0,C 180,E1 -28515.422,E2 -28515.422} C_VEL
LIN {X 0,Y 218.749,Z 768.756,A -85,B 0,C 180,E1 -28516.459,E2 -28516.459} C_VEL
LIN {X 0,Y 218.289,Z 779.042,A -85,B 0,C 180,E1 -28517.727,E2 -28517.727} C_VEL
LIN {X 0,Y 217.688,Z 788.193,A -85,B 0,C 180,E1 -28519.104,E2 -28519.104} C_VEL
LIN {X 0,Y 217.321,Z 796.104,A -85,B 0,C 180,E1 -28520.492,E2 -28520.492} C_VEL
LIN {X 0,Y 216.971,Z 804.034,A -85,B 0,C 180,E1 -28522.114,E2 -28522.114} C_VEL
LIN {X 0,Y 216.639,Z 813.436,A -85,B 0,C 180,E1 -28524.434,E2 -28524.434} C_VEL
LIN {X 0,Y 216.521,Z 819.859,A -85,B 0,C 180,E1 -28526.291,E2 -28526.291} C_VEL
LIN {X 0,Y 216.39,Z 826.582,A -85,B 0,C 180,E1 -28528.609,E2 -28528.609} C_VEL
LIN {X 0,Y 216.183,Z 832.149,A -85,B 0,C 180,E1 -28530.929,E2 -28530.929} C_VEL
LIN {X 0,Y 216,Z 835.162,A -85,B 0,C 180,E1 -28532.502,E2 -28532.502} C_VEL
LIN {X 0,Y 215.126,Z 837.547,A -85,B 0,C 180,E1 -28533.921,E2 -28533.921} C_VEL
LIN {X 0,Y 212.13,Z 840.47,A -85,B 0,C 180,E1 -28536.332,E2 -28536.332} C_VEL
LIN {X 0,Y 209.884,Z 842.378,A -85,B 0,C 180,E1 -28538.349,E2 -28538.349} C_VEL
LIN {X 0,Y 209.192,Z 843.829,A -85,B 0,C 180,E1 -28539.915,E2 -28539.915} C_VEL
LIN {X 0,Y 209.271,Z 844.294,A -85,B 0,C 180,E1 -28540.44,E2 -28540.44} C_VEL
LIN {X 0,Y 210.672,Z 846.823,A -85,B 0,C 180,E1 -28543.459,E2 -28543.459} C_VEL
LIN {X 0,Y 213.468,Z 848.72,A -85,B 0,C 180,E1 -28547.177,E2 -28547.177} C_VEL
LIN {X 0,Y 217.372,Z 849.146,A -85,B 0,C 180,E1 -28550.761,E2 -28550.761} C_VEL
LIN {X 0,Y 222.388,Z 848.1,A -85,B 0,C 180,E1 -28554.171,E2 -28554.171} C_VEL
LIN {X 0,Y 225.197,Z 847.058,A -85,B 0,C 180,E1 -28555.814,E2 -28555.814} C_VEL
LIN {X 0,Y 231.763,Z 843.915,A -85,B 0,C 180,E1 -28558.919,E2 -28558.919} C_VEL
LIN {X 0,Y 239.136,Z 839.081,A -85,B 0,C 180,E1 -28561.819,E2 -28561.819} C_VEL
LIN {X 0,Y 245.165,Z 834.334,A -85,B 0,C 180,E1 -28563.857,E2 -28563.857} C_VEL
LIN {X 0,Y 251.658,Z 828.495,A -85,B 0,C 180,E1 -28565.768,E2 -28565.768} C_VEL
LIN {X 0,Y 258.569,Z 821.362,A -85,B 0,C 180,E1 -28567.554,E2 -28567.554} C_VEL
LIN {X 0,Y 264.603,Z 814.265,A -85,B 0,C 180,E1 -28568.955,E2 -28568.955} C_VEL
LIN {X 0,Y 270.878,Z 805.836,A -85,B 0,C 180,E1 -28570.275,E2 -28570.275} C_VEL
LIN {X 0,Y 276.805,Z 796.942,A -85,B 0,C 180,E1 -28571.383,E2 -28571.383} C_VEL
LIN {X 0,Y 282.234,Z 787.565,A -85,B 0,C 180,E1 -28572.314,E2 -28572.314} C_VEL
LIN {X 0,Y 287.085,Z 777.829,A -85,B 0,C 180,E1 -28573.091,E2 -28573.091} C_VEL
LIN {X 0,Y 291.617,Z 767.018,A -85,B 0,C 180,E1 -28573.786,E2 -28573.786} C_VEL
LIN {X 0,Y 295.323,Z 756.447,A -85,B 0,C 180,E1 -28574.292,E2 -28574.292} C_VEL
LIN {X 0,Y 298.402,Z 745.536,A -85,B 0,C 180,E1 -28574.765,E2 -28574.765} C_VEL
LIN {X 0,Y 297.906,Z 742.68,A -85,B 0,C 180,E1 -28576.407,E2 -28576.407} C_VEL
LIN {X 0,Y 297.603,Z 739.523,A -85,B 0,C 180,E1 -28579.151,E2 -28579.151} C_VEL
LIN {X 0,Y 297.74,Z 739.374,A -85,B 0,C 180,E1 -28581.891,E2 -28581.891} C_VEL
LIN {X 0,Y 298.522,Z 741.744,A -85,B 0,C 180,E1 -28584.722,E2 -28584.722} C_VEL
LIN {X 0,Y 298.778,Z 743.067,A -85,B 0,C 180,E1 -28585.523,E2 -28585.523} C_VEL
LIN {X 0,Y 295.702,Z 753.969,A -85,B 0,C 180,E1 -28586.003,E2 -28586.003} C_VEL
LIN {X 0,Y 291.486,Z 765.96,A -85,B 0,C 180,E1 -28586.654,E2 -28586.654} C_VEL
LIN {X 0,Y 285.911,Z 778.827,A -85,B 0,C 180,E1 -28587.594,E2 -28587.594} C_VEL
LIN {X 0,Y 279.507,Z 790.642,A -85,B 0,C 180,E1 -28588.77,E2 -28588.77} C_VEL
LIN {X 0,Y 274.562,Z 798.529,A -85,B 0,C 180,E1 -28589.745,E2 -28589.745} C_VEL
LIN {X 0,Y 268.211,Z 807.393,A -85,B 0,C 180,E1 -28591.109,E2 -28591.109} C_VEL
LIN {X 0,Y 262.034,Z 814.939,A -85,B 0,C 180,E1 -28592.541,E2 -28592.541} C_VEL
LIN {X 0,Y 256.21,Z 821.21,A -85,B 0,C 180,E1 -28594.06,E2 -28594.06} C_VEL
LIN {X 0,Y 251.711,Z 825.585,A -85,B 0,C 180,E1 -28595.328,E2 -28595.328} C_VEL
LIN {X 0,Y 245.272,Z 831.002,A -85,B 0,C 180,E1 -28597.323,E2 -28597.323} C_VEL
LIN {X 0,Y 239.211,Z 835.322,A -85,B 0,C 180,E1 -28599.428,E2 -28599.428} C_VEL
LIN {X 0,Y 231.82,Z 839.375,A -85,B 0,C 180,E1 -28602.413,E2 -28602.413} C_VEL
LIN {X 0,Y 228.423,Z 840.883,A -85,B 0,C 180,E1 -28603.979,E2 -28603.979} C_VEL
LIN {X 0,Y 222.356,Z 842.582,A -85,B 0,C 180,E1 -28607.261,E2 -28607.261} C_VEL
LIN {X 0,Y 217.349,Z 842.686,A -85,B 0,C 180,E1 -28610.727,E2 -28610.727} C_VEL
LIN {X 0,Y 215.205,Z 842.264,A -85,B 0,C 180,E1 -28612.519,E2 -28612.519} C_VEL
LIN {X 0,Y 211.897,Z 840.2,A -85,B 0,C 180,E1 -28616.209,E2 -28616.209} C_VEL
LIN {X 0,Y 209.726,Z 836.565,A -85,B 0,C 180,E1 -28619.999,E2 -28619.999} C_VEL
LIN {X 0,Y 208.639,Z 832.562,A -85,B 0,C 180,E1 -28623.078,E2 -28623.078} C_VEL
LIN {X 0,Y 208.2,Z 828.094,A -85,B 0,C 180,E1 -28625.792,E2 -28625.792} C_VEL
LIN {X 0,Y 208.234,Z 822.187,A -85,B 0,C 180,E1 -28628.706,E2 -28628.706} C_VEL
LIN {X 0,Y 208.549,Z 814.877,A -85,B 0,C 180,E1 -28631.625,E2 -28631.625} C_VEL
LIN {X 0,Y 208.9,Z 807.457,A -85,B 0,C 180,E1 -28634.068,E2 -28634.068} C_VEL
LIN {X 0,Y 209.204,Z 799.344,A -85,B 0,C 180,E1 -28636.284,E2 -28636.284} C_VEL
LIN {X 0,Y 209.675,Z 790.762,A -85,B 0,C 180,E1 -28638.25,E2 -28638.25} C_VEL
LIN {X 0,Y 210.139,Z 781.21,A -85,B 0,C 180,E1 -28640.081,E2 -28640.081} C_VEL
LIN {X 0,Y 210.707,Z 771.032,A -85,B 0,C 180,E1 -28641.704,E2 -28641.704} C_VEL
LIN {X 0,Y 211.299,Z 760.741,A -85,B 0,C 180,E1 -28643.052,E2 -28643.052} C_VEL
LIN {X 0,Y 211.799,Z 750.242,A -85,B 0,C 180,E1 -28644.157,E2 -28644.157} C_VEL
LIN {X 0,Y 212.192,Z 738.778,A -85,B 0,C 180,E1 -28645.085,E2 -28645.085} C_VEL
LIN {X 0,Y 213.643,Z 693.574,A -85,B 0,C 180,E1 -28647.75,E2 -28647.75} C_VEL
LIN {X 0,Y 214.432,Z 666.486,A -85,B 0,C 180,E1 -28649.289,E2 -28649.289} C_VEL
LIN {X 0,Y 211.956,Z 638.785,A -85,B 0,C 180,E1 -28650.835,E2 -28650.835} C_VEL
LIN {X 0,Y 211.582,Z 631.068,A -85,B 0,C 180,E1 -28651.317,E2 -28651.317} C_VEL
LIN {X 0,Y 210.877,Z 631.142,A -85,B 0,C 180,E1 -28657.138,E2 -28657.138} C_VEL
LIN {X 0,Y 210.838,Z 631.155,A -85,B 0,C 180,E1 -28661.638,E2 -28661.638} C_VEL
LIN {X 0,Y 210.88,Z 631.145,A -85,B 0,C 180,E1 -28665.771,E2 -28665.771} C_VEL
LIN {X 0,Y 210.849,Z 631.152,A -85,B 0,C 180,E1 -28670.862,E2 -28670.862} C_VEL
LIN {X 0,Y 210.843,Z 631.149,A -85,B 0,C 180,E1 -28675.614,E2 -28675.614} C_VEL
LIN {X 0,Y 210.886,Z 631.15,A -85,B 0,C 180,E1 -28680.117,E2 -28680.117} C_VEL
LIN {X 0,Y 210.943,Z 631.136,A -85,B 0,C 180,E1 -28684.426,E2 -28684.426} C_VEL
LIN {X 0,Y 210.959,Z 631.138,A -85,B 0,C 180,E1 -28688.578,E2 -28688.578} C_VEL
LIN {X 0,Y 210.99,Z 631.133,A -85,B 0,C 180,E1 -28692.615,E2 -28692.615} C_VEL
LIN {X 0,Y 211.1,Z 631.118,A -85,B 0,C 180,E1 -28696.569,E2 -28696.569} C_VEL
LIN {X 0,Y 211.35,Z 631.088,A -85,B 0,C 180,E1 -28702.382,E2 -28702.382} C_VEL
LIN {X 0,Y 211.56,Z 631.061,A -85,B 0,C 180,E1 -28706.203,E2 -28706.203} C_VEL
LIN {X 0,Y 211.695,Z 631.05,A -85,B 0,C 180,E1 -28710,E2 -28710} C_VEL
LIN {X 0,Y 211.56,Z 631.061,A -85,B 0,C 180,E1 -28713.796,E2 -28713.796} C_VEL
LIN {X 0,Y 211.35,Z 631.088,A -85,B 0,C 180,E1 -28717.618,E2 -28717.618} C_VEL
LIN {X 0,Y 211.1,Z 631.118,A -85,B 0,C 180,E1 -28723.43,E2 -28723.43} C_VEL
LIN {X 0,Y 210.989,Z 631.133,A -85,B 0,C 180,E1 -28727.384,E2 -28727.384} C_VEL
LIN {X 0,Y 210.966,Z 631.138,A -85,B 0,C 180,E1 -28731.622,E2 -28731.622} C_VEL
LIN {X 0,Y 210.922,Z 631.143,A -85,B 0,C 180,E1 -28736.283,E2 -28736.283} C_VEL
LIN {X 0,Y 210.896,Z 631.147,A -85,B 0,C 180,E1 -28740.286,E2 -28740.286} C_VEL
LIN {X 0,Y 210.878,Z 631.145,A -85,B 0,C 180,E1 -28744.379,E2 -28744.379} C_VEL
LIN {X 0,Y 210.903,Z 631.144,A -85,B 0,C 180,E1 -28747.149,E2 -28747.149} C_VEL
LIN {X 0,Y 210.845,Z 631.152,A -85,B 0,C 180,E1 -28751.637,E2 -28751.637} C_VEL
LIN {X 0,Y 210.88,Z 631.146,A -85,B 0,C 180,E1 -28755.773,E2 -28755.773} C_VEL
LIN {X 0,Y 210.871,Z 631.147,A -85,B 0,C 180,E1 -28760.868,E2 -28760.868} C_VEL
LIN {X 0,Y 210.857,Z 631.148,A -85,B 0,C 180,E1 -28765.618,E2 -28765.618} C_VEL
LIN {X 0,Y 210.886,Z 631.148,A -85,B 0,C 180,E1 -28770.119,E2 -28770.119} C_VEL
LIN {X 0,Y 210.949,Z 631.137,A -85,B 0,C 180,E1 -28774.428,E2 -28774.428} C_VEL
LIN {X 0,Y 210.952,Z 631.139,A -85,B 0,C 180,E1 -28778.578,E2 -28778.578} C_VEL
LIN {X 0,Y 211.047,Z 631.126,A -85,B 0,C 180,E1 -28784.254,E2 -28784.254} C_VEL
LIN {X 0,Y 211.108,Z 631.12,A -85,B 0,C 180,E1 -28788.518,E2 -28788.518} C_VEL
LIN {X 0,Y 211.524,Z 631.062,A -85,B 0,C 180,E1 -28793.424,E2 -28793.424} C_VEL
LIN {X 0,Y 211.593,Z 631.061,A -85,B 0,C 180,E1 -28798.104,E2 -28798.104} C_VEL
LIN {X 0,Y 211.695,Z 631.047,A -85,B 0,C 180,E1 -28800.001,E2 -28800.001} C_VEL
LIN {X 0,Y 211.562,Z 631.06,A -85,B 0,C 180,E1 -28803.797,E2 -28803.797} C_VEL
LIN {X 0,Y 211.351,Z 631.091,A -85,B 0,C 180,E1 -28807.618,E2 -28807.618} C_VEL
LIN {X 0,Y 211.102,Z 631.117,A -85,B 0,C 180,E1 -28811.484,E2 -28811.484} C_VEL
LIN {X 0,Y 211.027,Z 631.13,A -85,B 0,C 180,E1 -28815.726,E2 -28815.726} C_VEL
LIN {X 0,Y 210.939,Z 631.137,A -85,B 0,C 180,E1 -28821.602,E2 -28821.602} C_VEL
LIN {X 0,Y 210.925,Z 631.144,A -85,B 0,C 180,E1 -28826.283,E2 -28826.283} C_VEL
LIN {X 0,Y 210.87,Z 631.146,A -85,B 0,C 180,E1 -28830.273,E2 -28830.273} C_VEL
LIN {X 0,Y 210.844,Z 631.153,A -85,B 0,C 180,E1 -28834.386,E2 -28834.386} C_VEL
LIN {X 0,Y 210.847,Z 631.15,A -85,B 0,C 180,E1 -28839.138,E2 -28839.138} C_VEL
LIN {X 0,Y 210.786,Z 631.161,A -85,B 0,C 180,E1 -28844.254,E2 -28844.254} C_VEL
LIN {X 0,Y 210.802,Z 631.157,A -85,B 0,C 180,E1 -28848.352,E2 -28848.352} C_VEL
LIN {X 0,Y 210.816,Z 631.153,A -85,B 0,C 180,E1 -28852.884,E2 -28852.884} C_VEL
LIN {X 0,Y 210.854,Z 631.153,A -85,B 0,C 180,E1 -28856.149,E2 -28856.149} C_VEL
LIN {X 0,Y 211.087,Z 631.122,A -85,B 0,C 180,E1 -28862.319,E2 -28862.319} C_VEL
LIN {X 0,Y 211.48,Z 631.199,A -85,B 0,C 180,E1 -28864.414,E2 -28864.414} C_VEL
LIN {X 0,Y 212.179,Z 635.01,A -85,B 0,C 180,E1 -28866.147,E2 -28866.147} C_VEL
LIN {X 0,Y 211.194,Z 640.635,A -85,B 0,C 180,E1 -28868.667,E2 -28868.667} C_VEL
LIN {X 0,Y 211.756,Z 660.656,A -85,B 0,C 180,E1 -28869.835,E2 -28869.835} C_VEL
LIN {X 0,Y 214.062,Z 691.698,A -85,B 0,C 180,E1 -28871.565,E2 -28871.565} C_VEL
LIN {X 0,Y 212.523,Z 746.572,A -85,B 0,C 180,E1 -28874.774,E2 -28874.774} C_VEL
LIN {X 0,Y 212.115,Z 757.947,A -85,B 0,C 180,E1 -28875.661,E2 -28875.661} C_VEL
LIN {X 0,Y 211.707,Z 768.457,A -85,B 0,C 180,E1 -28876.731,E2 -28876.731} C_VEL
LIN {X 0,Y 211.281,Z 778.765,A -85,B 0,C 180,E1 -28878.042,E2 -28878.042} C_VEL
LIN {X 0,Y 210.699,Z 787.922,A -85,B 0,C 180,E1 -28879.465,E2 -28879.465} C_VEL
LIN {X 0,Y 210.254,Z 796.983,A -85,B 0,C 180,E1 -28881.137,E2 -28881.137} C_VEL
LIN {X 0,Y 209.959,Z 804.746,A -85,B 0,C 180,E1 -28882.814,E2 -28882.814} C_VEL
LIN {X 0,Y 209.718,Z 812.335,A -85,B 0,C 180,E1 -28884.73,E2 -28884.73} C_VEL
LIN {X 0,Y 209.606,Z 820.284,A -85,B 0,C 180,E1 -28887.127,E2 -28887.127} C_VEL
LIN {X 0,Y 209.463,Z 826.778,A -85,B 0,C 180,E1 -28889.521,E2 -28889.521} C_VEL
LIN {X 0,Y 209.235,Z 832.166,A -85,B 0,C 180,E1 -28891.919,E2 -28891.919} C_VEL
LIN {X 0,Y 208.828,Z 837.329,A -85,B 0,C 180,E1 -28894.811,E2 -28894.811} C_VEL
LIN {X 0,Y 208.71,Z 841.423,A -85,B 0,C 180,E1 -28897.715,E2 -28897.715} C_VEL
LIN {X 0,Y 209.271,Z 844.294,A -85,B 0,C 180,E1 -28900.44,E2 -28900.44} C_VEL
LIN {X 0,Y 209.237,Z 845.652,A -85,B 0,C 180,E1 -28902.015,E2 -28902.015} C_VEL
LIN {X 0,Y 207.879,Z 847.1,A -85,B 0,C 180,E1 -28904.68,E2 -28904.68} C_VEL
LIN {X 0,Y 207.075,Z 847.838,A -85,B 0,C 180,E1 -28906.851,E2 -28906.851} C_VEL
LIN {X 0,Y 207.472,Z 848.387,A -85,B 0,C 180,E1 -28908.474,E2 -28908.474} C_VEL
LIN {X 0,Y 207.902,Z 848.474,A -85,B 0,C 180,E1 -28909.002,E2 -28909.002} C_VEL
LIN {X 0,Y 211.298,Z 848.921,A -85,B 0,C 180,E1 -28911.845,E2 -28911.845} C_VEL
LIN {X 0,Y 215.944,Z 848.307,A -85,B 0,C 180,E1 -28914.941,E2 -28914.941} C_VEL
LIN {X 0,Y 222.115,Z 846.295,A -85,B 0,C 180,E1 -28918.231,E2 -28918.231} C_VEL
LIN {X 0,Y 229.319,Z 842.702,A -85,B 0,C 180,E1 -28921.283,E2 -28921.283} C_VEL
LIN {X 0,Y 235.232,Z 839.009,A -85,B 0,C 180,E1 -28923.427,E2 -28923.427} C_VEL
LIN {X 0,Y 241.576,Z 834.395,A -85,B 0,C 180,E1 -28925.444,E2 -28925.444} C_VEL
LIN {X 0,Y 249.559,Z 827.483,A -85,B 0,C 180,E1 -28927.623,E2 -28927.623} C_VEL
LIN {X 0,Y 255.586,Z 821.511,A -85,B 0,C 180,E1 -28929.075,E2 -28929.075} C_VEL
LIN {X 0,Y 263.141,Z 812.983,A -85,B 0,C 180,E1 -28930.705,E2 -28930.705} C_VEL
LIN {X 0,Y 268.413,Z 806.326,A -85,B 0,C 180,E1 -28931.717,E2 -28931.717} C_VEL
LIN {X 0,Y 275.181,Z 796.409,A -85,B 0,C 180,E1 -28932.914,E2 -28932.914} C_VEL
LIN {X 0,Y 280.812,Z 786.872,A -85,B 0,C 180,E1 -28933.804,E2 -28933.804} C_VEL
LIN {X 0,Y 286.208,Z 776.313,A -85,B 0,C 180,E1 -28934.607,E2 -28934.607} C_VEL
LIN {X 0,Y 290.303,Z 766.917,A -85,B 0,C 180,E1 -28935.187,E2 -28935.187} C_VEL
LIN {X 0,Y 293.924,Z 757.141,A -85,B 0,C 180,E1 -28935.637,E2 -28935.637} C_VEL
LIN {X 0,Y 295.978,Z 750.705,A -85,B 0,C 180,E1 -28935.927,E2 -28935.927} C_VEL
LIN {X 0,Y 295.741,Z 748.828,A -85,B 0,C 180,E1 -28937.098,E2 -28937.098} C_VEL
LIN {X 0,Y 295.699,Z 746.329,A -85,B 0,C 180,E1 -28939.289,E2 -28939.289} C_VEL
LIN {X 0,Y 295.762,Z 746.157,A -85,B 0,C 180,E1 -28941.401,E2 -28941.401} C_VEL
LIN {X 0,Y 295.899,Z 746.782,A -85,B 0,C 180,E1 -28942.599,E2 -28942.599} C_VEL
LIN {X 0,Y 296.191,Z 747.745,A -85,B 0,C 180,E1 -28943.757,E2 -28943.757} C_VEL
LIN {X 0,Y 296.176,Z 749.162,A -85,B 0,C 180,E1 -28944.401,E2 -28944.401} C_VEL
LIN {X 0,Y 291.899,Z 761.788,A -85,B 0,C 180,E1 -28945.005,E2 -28945.005} C_VEL
LIN {X 0,Y 287.256,Z 772.835,A -85,B 0,C 180,E1 -28945.694,E2 -28945.694} C_VEL
LIN {X 0,Y 283.042,Z 781.379,A -85,B 0,C 180,E1 -28946.377,E2 -28946.377} C_VEL
LIN {X 0,Y 277.466,Z 791.218,A -85,B 0,C 180,E1 -28947.343,E2 -28947.343} C_VEL
LIN {X 0,Y 271.508,Z 800.28,A -85,B 0,C 180,E1 -28948.451,E2 -28948.451} C_VEL
LIN {X 0,Y 266.07,Z 807.519,A -85,B 0,C 180,E1 -28949.551,E2 -28949.551} C_VEL
LIN {X 0,Y 259.638,Z 814.977,A -85,B 0,C 180,E1 -28950.948,E2 -28950.948} C_VEL
LIN {X 0,Y 253.485,Z 821.333,A -85,B 0,C 180,E1 -28952.441,E2 -28952.441} C_VEL
LIN {X 0,Y 247.644,Z 826.658,A -85,B 0,C 180,E1 -28953.997,E2 -28953.997} C_VEL
LIN {X 0,Y 240.919,Z 831.874,A -85,B 0,C 180,E1 -28955.981,E2 -28955.981} C_VEL
LIN {X 0,Y 233.374,Z 836.654,A -85,B 0,C 180,E1 -28958.503,E2 -28958.503} C_VEL
LIN {X 0,Y 228.689,Z 839.172,A -85,B 0,C 180,E1 -28960.311,E2 -28960.311} C_VEL
LIN {X 0,Y 221.531,Z 841.823,A -85,B 0,C 180,E1 -28963.467,E2 -28963.467} C_VEL
LIN {X 0,Y 216.374,Z 842.88,A -85,B 0,C 180,E1 -28966.207,E2 -28966.207} C_VEL
LIN {X 0,Y 212.721,Z 843.045,A -85,B 0,C 180,E1 -28968.605,E2 -28968.605} C_VEL
LIN {X 0,Y 208.104,Z 841.888,A -85,B 0,C 180,E1 -28972.262,E2 -28972.262} C_VEL
LIN {X 0,Y 206.326,Z 840.849,A -85,B 0,C 180,E1 -28974.154,E2 -28974.154} C_VEL
LIN {X 0,Y 203.633,Z 837.568,A -85,B 0,C 180,E1 -28978.028,E2 -28978.028} C_VEL
LIN {X 0,Y 202.222,Z 834.054,A -85,B 0,C 180,E1 -28980.992,E2 -28980.992} C_VEL
LIN {X 0,Y 201.339,Z 827.829,A -85,B 0,C 180,E1 -28984.989,E2 -28984.989} C_VEL
LIN {X 0,Y 201.287,Z 821.889,A -85,B 0,C 180,E1 -28988,E2 -28988} C_VEL
LIN {X 0,Y 201.516,Z 815.906,A -85,B 0,C 180,E1 -28990.514,E2 -28990.514} C_VEL
LIN {X 0,Y 201.849,Z 808.535,A -85,B 0,C 180,E1 -28993.086,E2 -28993.086} C_VEL
LIN {X 0,Y 202.22,Z 799.93,A -85,B 0,C 180,E1 -28995.571,E2 -28995.571} C_VEL
LIN {X 0,Y 202.725,Z 790.402,A -85,B 0,C 180,E1 -28997.856,E2 -28997.856} C_VEL
LIN {X 0,Y 203.136,Z 781.495,A -85,B 0,C 180,E1 -28999.644,E2 -28999.644} C_VEL
LIN {X 0,Y 203.585,Z 772.427,A -85,B 0,C 180,E1 -29001.166,E2 -29001.166} C_VEL
LIN {X 0,Y 204.226,Z 761.313,A -85,B 0,C 180,E1 -29002.695,E2 -29002.695} C_VEL
LIN {X 0,Y 204.712,Z 750.942,A -85,B 0,C 180,E1 -29003.839,E2 -29003.839} C_VEL
LIN {X 0,Y 205.096,Z 739.692,A -85,B 0,C 180,E1 -29004.798,E2 -29004.798} C_VEL
LIN {X 0,Y 206.34,Z 703.033,A -85,B 0,C 180,E1 -29007.07,E2 -29007.07} C_VEL
LIN {X 0,Y 207.296,Z 666.606,A -85,B 0,C 180,E1 -29009.225,E2 -29009.225} C_VEL
LIN {X 0,Y 204.858,Z 638.612,A -85,B 0,C 180,E1 -29010.855,E2 -29010.855} C_VEL
LIN {X 0,Y 204.544,Z 631.945,A -85,B 0,C 180,E1 -29011.262,E2 -29011.262} C_VEL
LIN {X 0,Y 203.804,Z 632.029,A -85,B 0,C 180,E1 -29018.215,E2 -29018.215} C_VEL
LIN {X 0,Y 203.81,Z 632.029,A -85,B 0,C 180,E1 -29020.879,E2 -29020.879} C_VEL
LIN {X 0,Y 203.811,Z 632.03,A -85,B 0,C 180,E1 -29023.803,E2 -29023.803} C_VEL
LIN {X 0,Y 203.798,Z 632.025,A -85,B 0,C 180,E1 -29026.576,E2 -29026.576} C_VEL
LIN {X 0,Y 203.804,Z 632.028,A -85,B 0,C 180,E1 -29029.231,E2 -29029.231} C_VEL
LIN {X 0,Y 203.755,Z 632.033,A -85,B 0,C 180,E1 -29034.238,E2 -29034.238} C_VEL
LIN {X 0,Y 203.797,Z 632.029,A -85,B 0,C 180,E1 -29038.966,E2 -29038.966} C_VEL
LIN {X 0,Y 203.881,Z 632.019,A -85,B 0,C 180,E1 -29043.472,E2 -29043.472} C_VEL
LIN {X 0,Y 203.917,Z 632.015,A -85,B 0,C 180,E1 -29048.036,E2 -29048.036} C_VEL
LIN {X 0,Y 204.013,Z 632.001,A -85,B 0,C 180,E1 -29054.011,E2 -29054.011} C_VEL
LIN {X 0,Y 204.081,Z 631.996,A -85,B 0,C 180,E1 -29058.116,E2 -29058.116} C_VEL
LIN {X 0,Y 204.457,Z 631.946,A -85,B 0,C 180,E1 -29063.456,E2 -29063.456} C_VEL
LIN {X 0,Y 204.556,Z 631.937,A -85,B 0,C 180,E1 -29068.037,E2 -29068.037} C_VEL
LIN {X 0,Y 204.653,Z 631.927,A -85,B 0,C 180,E1 -29070,E2 -29070} C_VEL
LIN {X 0,Y 204.513,Z 631.938,A -85,B 0,C 180,E1 -29073.927,E2 -29073.927} C_VEL
LIN {X 0,Y 204.457,Z 631.946,A -85,B 0,C 180,E1 -29076.543,E2 -29076.543} C_VEL
LIN {X 0,Y 204.081,Z 631.996,A -85,B 0,C 180,E1 -29081.884,E2 -29081.884} C_VEL
LIN {X 0,Y 204.013,Z 632.001,A -85,B 0,C 180,E1 -29085.988,E2 -29085.988} C_VEL
LIN {X 0,Y 203.916,Z 632.015,A -85,B 0,C 180,E1 -29091.963,E2 -29091.963} C_VEL
LIN {X 0,Y 203.863,Z 632.021,A -85,B 0,C 180,E1 -29096.708,E2 -29096.708} C_VEL
LIN {X 0,Y 203.833,Z 632.024,A -85,B 0,C 180,E1 -29101.027,E2 -29101.027} C_VEL
LIN {X 0,Y 203.815,Z 632.025,A -85,B 0,C 180,E1 -29105.749,E2 -29105.749} C_VEL
LIN {X 0,Y 203.817,Z 632.03,A -85,B 0,C 180,E1 -29108.213,E2 -29108.213} C_VEL
LIN {X 0,Y 203.807,Z 632.027,A -85,B 0,C 180,E1 -29110.88,E2 -29110.88} C_VEL
LIN {X 0,Y 203.812,Z 632.024,A -85,B 0,C 180,E1 -29113.805,E2 -29113.805} C_VEL
LIN {X 0,Y 203.802,Z 632.029,A -85,B 0,C 180,E1 -29116.578,E2 -29116.578} C_VEL
LIN {X 0,Y 203.802,Z 632.03,A -85,B 0,C 180,E1 -29119.232,E2 -29119.232} C_VEL
LIN {X 0,Y 203.813,Z 632.024,A -85,B 0,C 180,E1 -29122.226,E2 -29122.226} C_VEL
LIN {X 0,Y 203.797,Z 632.03,A -85,B 0,C 180,E1 -29126.64,E2 -29126.64} C_VEL
LIN {X 0,Y 203.822,Z 632.025,A -85,B 0,C 180,E1 -29131.242,E2 -29131.242} C_VEL
LIN {X 0,Y 203.881,Z 632.014,A -85,B 0,C 180,E1 -29133.474,E2 -29133.474} C_VEL
LIN {X 0,Y 203.869,Z 632.024,A -85,B 0,C 180,E1 -29138.071,E2 -29138.071} C_VEL
LIN {X 0,Y 203.91,Z 632.012,A -85,B 0,C 180,E1 -29141.992,E2 -29141.992} C_VEL
LIN {X 0,Y 204.004,Z 632.006,A -85,B 0,C 180,E1 -29146.094,E2 -29146.094} C_VEL
LIN {X 0,Y 204.134,Z 631.988,A -85,B 0,C 180,E1 -29150.122,E2 -29150.122} C_VEL
LIN {X 0,Y 204.466,Z 631.945,A -85,B 0,C 180,E1 -29154.102,E2 -29154.102} C_VEL
LIN {X 0,Y 204.56,Z 631.938,A -85,B 0,C 180,E1 -29158.038,E2 -29158.038} C_VEL
LIN {X 0,Y 204.653,Z 631.924,A -85,B 0,C 180,E1 -29160.001,E2 -29160.001} C_VEL
LIN {X 0,Y 204.515,Z 631.938,A -85,B 0,C 180,E1 -29163.928,E2 -29163.928} C_VEL
LIN {X 0,Y 204.46,Z 631.948,A -85,B 0,C 180,E1 -29166.544,E2 -29166.544} C_VEL
LIN {X 0,Y 204.042,Z 631.996,A -85,B 0,C 180,E1 -29171.887,E2 -29171.887} C_VEL
LIN {X 0,Y 203.972,Z 632.01,A -85,B 0,C 180,E1 -29175.946,E2 -29175.946} C_VEL
LIN {X 0,Y 203.869,Z 632.017,A -85,B 0,C 180,E1 -29181.929,E2 -29181.929} C_VEL
LIN {X 0,Y 203.866,Z 632.022,A -85,B 0,C 180,E1 -29186.709,E2 -29186.709} C_VEL
LIN {X 0,Y 203.799,Z 632.024,A -85,B 0,C 180,E1 -29191.034,E2 -29191.034} C_VEL
LIN {X 0,Y 203.755,Z 632.037,A -85,B 0,C 180,E1 -29195.761,E2 -29195.761} C_VEL
LIN {X 0,Y 203.782,Z 632.032,A -85,B 0,C 180,E1 -29198.222,E2 -29198.222} C_VEL
LIN {X 0,Y 203.779,Z 632.026,A -85,B 0,C 180,E1 -29200.87,E2 -29200.87} C_VEL
LIN {X 0,Y 203.73,Z 632.041,A -85,B 0,C 180,E1 -29206.221,E2 -29206.221} C_VEL
LIN {X 0,Y 203.769,Z 632.031,A -85,B 0,C 180,E1 -29209.224,E2 -29209.224} C_VEL
LIN {X 0,Y 203.775,Z 632.031,A -85,B 0,C 180,E1 -29212.241,E2 -29212.241} C_VEL
LIN {X 0,Y 203.788,Z 632.031,A -85,B 0,C 180,E1 -29216.638,E2 -29216.638} C_VEL
LIN {X 0,Y 203.938,Z 632.006,A -85,B 0,C 180,E1 -29221.26,E2 -29221.26} C_VEL
LIN {X 0,Y 204.485,Z 632.096,A -85,B 0,C 180,E1 -29224.716,E2 -29224.716} C_VEL
LIN {X 0,Y 205.018,Z 635.538,A -85,B 0,C 180,E1 -29226.333,E2 -29226.333} C_VEL
LIN {X 0,Y 204.11,Z 640.578,A -85,B 0,C 180,E1 -29228.682,E2 -29228.682} C_VEL
LIN {X 0,Y 204.675,Z 660.931,A -85,B 0,C 180,E1 -29229.89,E2 -29229.89} C_VEL
LIN {X 0,Y 206.992,Z 691.336,A -85,B 0,C 180,E1 -29231.659,E2 -29231.659} C_VEL
LIN {X 0,Y 205.489,Z 746.303,A -85,B 0,C 180,E1 -29234.999,E2 -29234.999} C_VEL
LIN {X 0,Y 205.081,Z 757.658,A -85,B 0,C 180,E1 -29235.916,E2 -29235.916} C_VEL
LIN {X 0,Y 204.681,Z 768.164,A -85,B 0,C 180,E1 -29237.022,E2 -29237.022} C_VEL
LIN {X 0,Y 204.276,Z 778.482,A -85,B 0,C 180,E1 -29238.379,E2 -29238.379} C_VEL
LIN {X 0,Y 203.712,Z 787.646,A -85,B 0,C 180,E1 -29239.851,E2 -29239.851} C_VEL
LIN {X 0,Y 203.284,Z 796.711,A -85,B 0,C 180,E1 -29241.58,E2 -29241.58} C_VEL
LIN {X 0,Y 203.034,Z 803.459,A -85,B 0,C 180,E1 -29243.065,E2 -29243.065} C_VEL
LIN {X 0,Y 202.832,Z 812.776,A -85,B 0,C 180,E1 -29245.544,E2 -29245.544} C_VEL
LIN {X 0,Y 202.74,Z 820.492,A -85,B 0,C 180,E1 -29248.02,E2 -29248.02} C_VEL
LIN {X 0,Y 202.561,Z 826.866,A -85,B 0,C 180,E1 -29250.496,E2 -29250.496} C_VEL
LIN {X 0,Y 202.236,Z 832.143,A -85,B 0,C 180,E1 -29252.978,E2 -29252.978} C_VEL
LIN {X 0,Y 201.898,Z 837.245,A -85,B 0,C 180,E1 -29255.974,E2 -29255.974} C_VEL
LIN {X 0,Y 202.136,Z 842.271,A -85,B 0,C 180,E1 -29259.978,E2 -29259.978} C_VEL
LIN {X 0,Y 202.805,Z 844.32,A -85,B 0,C 180,E1 -29261.96,E2 -29261.96} C_VEL
LIN {X 0,Y 205.009,Z 847.248,A -85,B 0,C 180,E1 -29265.863,E2 -29265.863} C_VEL
LIN {X 0,Y 207.902,Z 848.474,A -85,B 0,C 180,E1 -29269.002,E2 -29269.002} C_VEL
LIN {X 0,Y 208.932,Z 848.872,A -85,B 0,C 180,E1 -29270.603,E2 -29270.603} C_VEL
LIN {X 0,Y 209.412,Z 849.019,A -85,B 0,C 180,E1 -29273.324,E2 -29273.324} C_VEL
LIN {X 0,Y 210.551,Z 848.455,A -85,B 0,C 180,E1 -29275.998,E2 -29275.998} C_VEL
LIN {X 0,Y 212.556,Z 847.741,A -85,B 0,C 180,E1 -29277.483,E2 -29277.483} C_VEL
LIN {X 0,Y 219.516,Z 845.344,A -85,B 0,C 180,E1 -29280.7,E2 -29280.7} C_VEL
LIN {X 0,Y 226.426,Z 842.006,A -85,B 0,C 180,E1 -29283.359,E2 -29283.359} C_VEL
LIN {X 0,Y 231.553,Z 839.065,A -85,B 0,C 180,E1 -29285.082,E2 -29285.082} C_VEL
LIN {X 0,Y 238.228,Z 834.475,A -85,B 0,C 180,E1 -29287.067,E2 -29287.067} C_VEL
LIN {X 0,Y 246.558,Z 827.658,A -85,B 0,C 180,E1 -29289.206,E2 -29289.206} C_VEL
LIN {X 0,Y 254.084,Z 820.539,A -85,B 0,C 180,E1 -29290.899,E2 -29290.899} C_VEL
LIN {X 0,Y 260.66,Z 813.422,A -85,B 0,C 180,E1 -29292.207,E2 -29292.207} C_VEL
LIN {X 0,Y 267.485,Z 804.921,A -85,B 0,C 180,E1 -29293.424,E2 -29293.424} C_VEL
LIN {X 0,Y 274.049,Z 795.666,A -85,B 0,C 180,E1 -29294.479,E2 -29294.479} C_VEL
LIN {X 0,Y 279.622,Z 786.617,A -85,B 0,C 180,E1 -29295.292,E2 -29295.292} C_VEL
LIN {X 0,Y 284.881,Z 776.643,A -85,B 0,C 180,E1 -29296.017,E2 -29296.017} C_VEL
LIN {X 0,Y 289.238,Z 766.895,A -85,B 0,C 180,E1 -29296.595,E2 -29296.595} C_VEL
LIN {X 0,Y 293.014,Z 756.862,A -85,B 0,C 180,E1 -29297.043,E2 -29297.043} C_VEL
LIN {X 0,Y 293.379,Z 755.593,A -85,B 0,C 180,E1 -29297.172,E2 -29297.172} C_VEL
LIN {X 0,Y 293.478,Z 752.979,A -85,B 0,C 180,E1 -29299.878,E2 -29299.878} C_VEL
LIN {X 0,Y 293.67,Z 753.035,A -85,B 0,C 180,E1 -29301.916,E2 -29301.916} C_VEL
LIN {X 0,Y 293.695,Z 754.029,A -85,B 0,C 180,E1 -29303.191,E2 -29303.191} C_VEL
LIN {X 0,Y 289.834,Z 764.623,A -85,B 0,C 180,E1 -29303.751,E2 -29303.751} C_VEL
LIN {X 0,Y 285.016,Z 775.416,A -85,B 0,C 180,E1 -29304.423,E2 -29304.423} C_VEL
LIN {X 0,Y 279.654,Z 785.506,A -85,B 0,C 180,E1 -29305.262,E2 -29305.262} C_VEL
LIN {X 0,Y 272.503,Z 796.838,A -85,B 0,C 180,E1 -29306.451,E2 -29306.451} C_VEL
LIN {X 0,Y 264.175,Z 807.687,A -85,B 0,C 180,E1 -29307.975,E2 -29307.975} C_VEL
LIN {X 0,Y 257.493,Z 815.21,A -85,B 0,C 180,E1 -29309.333,E2 -29309.333} C_VEL
LIN {X 0,Y 251.04,Z 821.528,A -85,B 0,C 180,E1 -29310.772,E2 -29310.772} C_VEL
LIN {X 0,Y 243.717,Z 827.717,A -85,B 0,C 180,E1 -29312.623,E2 -29312.623} C_VEL
LIN {X 0,Y 239.004,Z 831.329,A -85,B 0,C 180,E1 -29313.921,E2 -29313.921} C_VEL
LIN {X 0,Y 232.226,Z 835.655,A -85,B 0,C 180,E1 -29315.971,E2 -29315.971} C_VEL
LIN {X 0,Y 225.885,Z 838.923,A -85,B 0,C 180,E1 -29318.154,E2 -29318.154} C_VEL
LIN {X 0,Y 218.189,Z 841.815,A -85,B 0,C 180,E1 -29321.274,E2 -29321.274} C_VEL
LIN {X 0,Y 211.365,Z 843.13,A -85,B 0,C 180,E1 -29324.626,E2 -29324.626} C_VEL
LIN {X 0,Y 208.391,Z 843.326,A -85,B 0,C 180,E1 -29326.391,E2 -29326.391} C_VEL
LIN {X 0,Y 203.198,Z 842.433,A -85,B 0,C 180,E1 -29330.075,E2 -29330.075} C_VEL
LIN {X 0,Y 199.237,Z 840.042,A -85,B 0,C 180,E1 -29333.945,E2 -29333.945} C_VEL
LIN {X 0,Y 197.099,Z 837.386,A -85,B 0,C 180,E1 -29336.944,E2 -29336.944} C_VEL
LIN {X 0,Y 195.579,Z 833.828,A -85,B 0,C 180,E1 -29339.999,E2 -29339.999} C_VEL
LIN {X 0,Y 194.673,Z 829.288,A -85,B 0,C 180,E1 -29343.093,E2 -29343.093} C_VEL
LIN {X 0,Y 194.34,Z 822.602,A -85,B 0,C 180,E1 -29346.726,E2 -29346.726} C_VEL
LIN {X 0,Y 194.569,Z 815.534,A -85,B 0,C 180,E1 -29349.845,E2 -29349.845} C_VEL
LIN {X 0,Y 194.903,Z 808.281,A -85,B 0,C 180,E1 -29352.452,E2 -29352.452} C_VEL
LIN {X 0,Y 195.241,Z 800.444,A -85,B 0,C 180,E1 -29354.809,E2 -29354.809} C_VEL
LIN {X 0,Y 195.699,Z 791.01,A -85,B 0,C 180,E1 -29357.174,E2 -29357.174} C_VEL
LIN {X 0,Y 196.107,Z 782.239,A -85,B 0,C 180,E1 -29359.021,E2 -29359.021} C_VEL
LIN {X 0,Y 196.604,Z 771.647,A -85,B 0,C 180,E1 -29360.871,E2 -29360.871} C_VEL
LIN {X 0,Y 197.179,Z 761.43,A -85,B 0,C 180,E1 -29362.34,E2 -29362.34} C_VEL
LIN {X 0,Y 197.666,Z 751.58,A -85,B 0,C 180,E1 -29363.493,E2 -29363.493} C_VEL
LIN {X 0,Y 198,Z 740.605,A -85,B 0,C 180,E1 -29364.491,E2 -29364.491} C_VEL
LIN {X 0,Y 198.973,Z 711.61,A -85,B 0,C 180,E1 -29366.387,E2 -29366.387} C_VEL
LIN {X 0,Y 200.263,Z 667.417,A -85,B 0,C 180,E1 -29369.111,E2 -29369.111} C_VEL
LIN {X 0,Y 197.778,Z 639.005,A -85,B 0,C 180,E1 -29370.828,E2 -29370.828} C_VEL
LIN {X 0,Y 197.5,Z 632.822,A -85,B 0,C 180,E1 -29371.232,E2 -29371.232} C_VEL
LIN {X 0,Y 196.761,Z 632.906,A -85,B 0,C 180,E1 -29378.447,E2 -29378.447} C_VEL
LIN {X 0,Y 196.722,Z 632.911,A -85,B 0,C 180,E1 -29382.57,E2 -29382.57} C_VEL
LIN {X 0,Y 196.722,Z 632.907,A -85,B 0,C 180,E1 -29387.428,E2 -29387.428} C_VEL
LIN {X 0,Y 196.744,Z 632.91,A -85,B 0,C 180,E1 -29391.557,E2 -29391.557} C_VEL
LIN {X 0,Y 196.739,Z 632.904,A -85,B 0,C 180,E1 -29395.274,E2 -29395.274} C_VEL
LIN {X 0,Y 196.737,Z 632.913,A -85,B 0,C 180,E1 -29400.102,E2 -29400.102} C_VEL
LIN {X 0,Y 196.801,Z 632.896,A -85,B 0,C 180,E1 -29404.716,E2 -29404.716} C_VEL
LIN {X 0,Y 196.836,Z 632.896,A -85,B 0,C 180,E1 -29409.154,E2 -29409.154} C_VEL
LIN {X 0,Y 196.96,Z 632.881,A -85,B 0,C 180,E1 -29413.776,E2 -29413.776} C_VEL
LIN {X 0,Y 197.012,Z 632.873,A -85,B 0,C 180,E1 -29417.683,E2 -29417.683} C_VEL
LIN {X 0,Y 197.418,Z 632.823,A -85,B 0,C 180,E1 -29423.43,E2 -29423.43} C_VEL
LIN {X 0,Y 197.523,Z 632.812,A -85,B 0,C 180,E1 -29427.967,E2 -29427.967} C_VEL
LIN {X 0,Y 197.613,Z 632.804,A -85,B 0,C 180,E1 -29430,E2 -29430} C_VEL
LIN {X 0,Y 197.47,Z 632.814,A -85,B 0,C 180,E1 -29434.068,E2 -29434.068} C_VEL
LIN {X 0,Y 197.417,Z 632.823,A -85,B 0,C 180,E1 -29436.57,E2 -29436.57} C_VEL
LIN {X 0,Y 197.012,Z 632.874,A -85,B 0,C 180,E1 -29442.317,E2 -29442.317} C_VEL
LIN {X 0,Y 196.939,Z 632.883,A -85,B 0,C 180,E1 -29446.531,E2 -29446.531} C_VEL
LIN {X 0,Y 196.844,Z 632.894,A -85,B 0,C 180,E1 -29452.307,E2 -29452.307} C_VEL
LIN {X 0,Y 196.78,Z 632.904,A -85,B 0,C 180,E1 -29457.564,E2 -29457.564} C_VEL
LIN {X 0,Y 196.751,Z 632.905,A -85,B 0,C 180,E1 -29462.276,E2 -29462.276} C_VEL
LIN {X 0,Y 196.768,Z 632.901,A -85,B 0,C 180,E1 -29465.043,E2 -29465.043} C_VEL
LIN {X 0,Y 196.727,Z 632.913,A -85,B 0,C 180,E1 -29469.858,E2 -29469.858} C_VEL
LIN {X 0,Y 196.728,Z 632.907,A -85,B 0,C 180,E1 -29474.596,E2 -29474.596} C_VEL
LIN {X 0,Y 196.729,Z 632.912,A -85,B 0,C 180,E1 -29478.391,E2 -29478.391} C_VEL
LIN {X 0,Y 196.745,Z 632.903,A -85,B 0,C 180,E1 -29482.756,E2 -29482.756} C_VEL
LIN {X 0,Y 196.775,Z 632.901,A -85,B 0,C 180,E1 -29485.283,E2 -29485.283} C_VEL
LIN {X 0,Y 196.737,Z 632.91,A -85,B 0,C 180,E1 -29490.104,E2 -29490.104} C_VEL
LIN {X 0,Y 196.802,Z 632.899,A -85,B 0,C 180,E1 -29494.717,E2 -29494.717} C_VEL
LIN {X 0,Y 196.808,Z 632.901,A -85,B 0,C 180,E1 -29499.152,E2 -29499.152} C_VEL
LIN {X 0,Y 196.924,Z 632.881,A -85,B 0,C 180,E1 -29503.814,E2 -29503.814} C_VEL
LIN {X 0,Y 196.981,Z 632.881,A -85,B 0,C 180,E1 -29507.682,E2 -29507.682} C_VEL
LIN {X 0,Y 197.42,Z 632.818,A -85,B 0,C 180,E1 -29513.431,E2 -29513.431} C_VEL
LIN {X 0,Y 197.528,Z 632.814,A -85,B 0,C 180,E1 -29517.968,E2 -29517.968} C_VEL
LIN {X 0,Y 197.613,Z 632.8,A -85,B 0,C 180,E1 -29520.001,E2 -29520.001} C_VEL
LIN {X 0,Y 197.473,Z 632.816,A -85,B 0,C 180,E1 -29524.069,E2 -29524.069} C_VEL
LIN {X 0,Y 197.42,Z 632.825,A -85,B 0,C 180,E1 -29526.57,E2 -29526.57} C_VEL
LIN {X 0,Y 196.973,Z 632.876,A -85,B 0,C 180,E1 -29532.32,E2 -29532.32} C_VEL
LIN {X 0,Y 196.87,Z 632.894,A -85,B 0,C 180,E1 -29536.537,E2 -29536.537} C_VEL
LIN {X 0,Y 196.804,Z 632.897,A -85,B 0,C 180,E1 -29542.278,E2 -29542.278} C_VEL
LIN {X 0,Y 196.799,Z 632.902,A -85,B 0,C 180,E1 -29547.153,E2 -29547.153} C_VEL
LIN {X 0,Y 196.726,Z 632.908,A -85,B 0,C 180,E1 -29552.282,E2 -29552.282} C_VEL
LIN {X 0,Y 196.729,Z 632.91,A -85,B 0,C 180,E1 -29555.025,E2 -29555.025} C_VEL
LIN {X 0,Y 196.697,Z 632.913,A -85,B 0,C 180,E1 -29559.866,E2 -29559.866} C_VEL
LIN {X 0,Y 196.649,Z 632.921,A -85,B 0,C 180,E1 -29564.572,E2 -29564.572} C_VEL
LIN {X 0,Y 196.695,Z 632.914,A -85,B 0,C 180,E1 -29568.403,E2 -29568.403} C_VEL
LIN {X 0,Y 196.712,Z 632.91,A -85,B 0,C 180,E1 -29572.748,E2 -29572.748} C_VEL
LIN {X 0,Y 196.736,Z 632.911,A -85,B 0,C 180,E1 -29577.721,E2 -29577.721} C_VEL
LIN {X 0,Y 197.494,Z 632.878,A -85,B 0,C 180,E1 -29585.022,E2 -29585.022} C_VEL
LIN {X 0,Y 197.893,Z 634.847,A -85,B 0,C 180,E1 -29585.981,E2 -29585.981} C_VEL
LIN {X 0,Y 197.014,Z 640.38,A -85,B 0,C 180,E1 -29588.655,E2 -29588.655} C_VEL
LIN {X 0,Y 197.653,Z 662.764,A -85,B 0,C 180,E1 -29590.064,E2 -29590.064} C_VEL
LIN {X 0,Y 199.915,Z 691.347,A -85,B 0,C 180,E1 -29591.784,E2 -29591.784} C_VEL
LIN {X 0,Y 198.456,Z 746.012,A -85,B 0,C 180,E1 -29595.24,E2 -29595.24} C_VEL
LIN {X 0,Y 198.052,Z 757.355,A -85,B 0,C 180,E1 -29596.189,E2 -29596.189} C_VEL
LIN {X 0,Y 197.653,Z 767.86,A -85,B 0,C 180,E1 -29597.334,E2 -29597.334} C_VEL
LIN {X 0,Y 197.282,Z 778.107,A -85,B 0,C 180,E1 -29598.74,E2 -29598.74} C_VEL
LIN {X 0,Y 196.731,Z 788.58,A -85,B 0,C 180,E1 -29600.522,E2 -29600.522} C_VEL
LIN {X 0,Y 196.358,Z 797.349,A -85,B 0,C 180,E1 -29602.313,E2 -29602.313} C_VEL
LIN {X 0,Y 196.09,Z 805.841,A -85,B 0,C 180,E1 -29604.363,E2 -29604.363} C_VEL
LIN {X 0,Y 195.968,Z 813.088,A -85,B 0,C 180,E1 -29606.414,E2 -29606.414} C_VEL
LIN {X 0,Y 195.888,Z 819.331,A -85,B 0,C 180,E1 -29608.464,E2 -29608.464} C_VEL
LIN {X 0,Y 195.697,Z 825.843,A -85,B 0,C 180,E1 -29611.026,E2 -29611.026} C_VEL
LIN {X 0,Y 195.261,Z 832.058,A -85,B 0,C 180,E1 -29614.115,E2 -29614.115} C_VEL
LIN {X 0,Y 194.955,Z 836.997,A -85,B 0,C 180,E1 -29617.224,E2 -29617.224} C_VEL
LIN {X 0,Y 195.616,Z 842.051,A -85,B 0,C 180,E1 -29621.358,E2 -29621.358} C_VEL
LIN {X 0,Y 197.007,Z 844.933,A -85,B 0,C 180,E1 -29624.412,E2 -29624.412} C_VEL
LIN {X 0,Y 199.997,Z 847.406,A -85,B 0,C 180,E1 -29628.374,E2 -29628.374} C_VEL
LIN {X 0,Y 201.876,Z 848.201,A -85,B 0,C 180,E1 -29630.302,E2 -29630.302} C_VEL
LIN {X 0,Y 206.673,Z 848.695,A -85,B 0,C 180,E1 -29633.998,E2 -29633.998} C_VEL
LIN {X 0,Y 212.556,Z 847.741,A -85,B 0,C 180,E1 -29637.483,E2 -29637.483} C_VEL
LIN {X 0,Y 214.776,Z 846.919,A -85,B 0,C 180,E1 -29638.936,E2 -29638.936} C_VEL
LIN {X 0,Y 217.21,Z 845.477,A -85,B 0,C 180,E1 -29641.459,E2 -29641.459} C_VEL
LIN {X 0,Y 220.074,Z 843.548,A -85,B 0,C 180,E1 -29643.882,E2 -29643.882} C_VEL
LIN {X 0,Y 222.885,Z 841.907,A -85,B 0,C 180,E1 -29645.149,E2 -29645.149} C_VEL
LIN {X 0,Y 228.103,Z 839.1,A -85,B 0,C 180,E1 -29646.784,E2 -29646.784} C_VEL
LIN {X 0,Y 235.081,Z 834.614,A -85,B 0,C 180,E1 -29648.735,E2 -29648.735} C_VEL
LIN {X 0,Y 243.784,Z 827.972,A -85,B 0,C 180,E1 -29650.818,E2 -29650.818} C_VEL
LIN {X 0,Y 251.622,Z 820.886,A -85,B 0,C 180,E1 -29652.459,E2 -29652.459} C_VEL
LIN {X 0,Y 259.779,Z 812.359,A -85,B 0,C 180,E1 -29653.972,E2 -29653.972} C_VEL
LIN {X 0,Y 266.87,Z 803.84,A -85,B 0,C 180,E1 -29655.126,E2 -29655.126} C_VEL
LIN {X 0,Y 272.696,Z 795.82,A -85,B 0,C 180,E1 -29655.989,E2 -29655.989} C_VEL
LIN {X 0,Y 278.67,Z 786.328,A -85,B 0,C 180,E1 -29656.797,E2 -29656.797} C_VEL
LIN {X 0,Y 283.946,Z 776.638,A -85,B 0,C 180,E1 -29657.474,E2 -29657.474} C_VEL
LIN {X 0,Y 288.663,Z 766.531,A -85,B 0,C 180,E1 -29658.031,E2 -29658.031} C_VEL
LIN {X 0,Y 290.91,Z 761.132,A -85,B 0,C 180,E1 -29658.281,E2 -29658.281} C_VEL
LIN {X 0,Y 291.043,Z 760.052,A -85,B 0,C 180,E1 -29659.473,E2 -29659.473} C_VEL
LIN {X 0,Y 291.075,Z 759.64,A -85,B 0,C 180,E1 -29660.359,E2 -29660.359} C_VEL
LIN {X 0,Y 291.186,Z 759.662,A -85,B 0,C 180,E1 -29661.286,E2 -29661.286} C_VEL
LIN {X 0,Y 291.184,Z 760.06,A -85,B 0,C 180,E1 -29662.094,E2 -29662.094} C_VEL
LIN {X 0,Y 285.752,Z 772.441,A -85,B 0,C 180,E1 -29662.769,E2 -29662.769} C_VEL
LIN {X 0,Y 280.835,Z 781.799,A -85,B 0,C 180,E1 -29663.431,E2 -29663.431} C_VEL
LIN {X 0,Y 274.841,Z 791.724,A -85,B 0,C 180,E1 -29664.339,E2 -29664.339} C_VEL
LIN {X 0,Y 269.706,Z 799.123,A -85,B 0,C 180,E1 -29665.155,E2 -29665.155} C_VEL
LIN {X 0,Y 263.984,Z 806.4,A -85,B 0,C 180,E1 -29666.137,E2 -29666.137} C_VEL
LIN {X 0,Y 256.998,Z 814.073,A -85,B 0,C 180,E1 -29667.433,E2 -29667.433} C_VEL
LIN {X 0,Y 248.871,Z 821.794,A -85,B 0,C 180,E1 -29669.093,E2 -29669.093} C_VEL
LIN {X 0,Y 240.973,Z 828.178,A -85,B 0,C 180,E1 -29670.956,E2 -29670.956} C_VEL
LIN {X 0,Y 235.027,Z 832.305,A -85,B 0,C 180,E1 -29672.487,E2 -29672.487} C_VEL
LIN {X 0,Y 227.961,Z 836.453,A -85,B 0,C 180,E1 -29674.521,E2 -29674.521} C_VEL
LIN {X 0,Y 220.9,Z 839.767,A -85,B 0,C 180,E1 -29676.862,E2 -29676.862} C_VEL
LIN {X 0,Y 215.225,Z 841.798,A -85,B 0,C 180,E1 -29679.023,E2 -29679.023} C_VEL
LIN {X 0,Y 207.779,Z 843.305,A -85,B 0,C 180,E1 -29682.338,E2 -29682.338} C_VEL
LIN {X 0,Y 203.337,Z 843.561,A -85,B 0,C 180,E1 -29684.695,E2 -29684.695} C_VEL
LIN {X 0,Y 198.657,Z 842.891,A -85,B 0,C 180,E1 -29687.786,E2 -29687.786} C_VEL
LIN {X 0,Y 193.953,Z 840.754,A -85,B 0,C 180,E1 -29691.694,E2 -29691.694} C_VEL
LIN {X 0,Y 190.666,Z 837.13,A -85,B 0,C 180,E1 -29695.786,E2 -29695.786} C_VEL
LIN {X 0,Y 189.181,Z 834.024,A -85,B 0,C 180,E1 -29698.568,E2 -29698.568} C_VEL
LIN {X 0,Y 187.933,Z 828.924,A -85,B 0,C 180,E1 -29702.135,E2 -29702.135} C_VEL
LIN {X 0,Y 187.493,Z 822.124,A -85,B 0,C 180,E1 -29705.896,E2 -29705.896} C_VEL
LIN {X 0,Y 187.646,Z 816.335,A -85,B 0,C 180,E1 -29708.586,E2 -29708.586} C_VEL
LIN {X 0,Y 187.897,Z 809.389,A -85,B 0,C 180,E1 -29711.285,E2 -29711.285} C_VEL
LIN {X 0,Y 188.286,Z 801.511,A -85,B 0,C 180,E1 -29713.841,E2 -29713.841} C_VEL
LIN {X 0,Y 188.661,Z 791.584,A -85,B 0,C 180,E1 -29716.444,E2 -29716.444} C_VEL
LIN {X 0,Y 189.152,Z 781.553,A -85,B 0,C 180,E1 -29718.625,E2 -29718.625} C_VEL
LIN {X 0,Y 189.563,Z 772.535,A -85,B 0,C 180,E1 -29720.267,E2 -29720.267} C_VEL
LIN {X 0,Y 190.178,Z 761.42,A -85,B 0,C 180,E1 -29721.933,E2 -29721.933} C_VEL
LIN {X 0,Y 190.671,Z 750.9,A -85,B 0,C 180,E1 -29723.196,E2 -29723.196} C_VEL
LIN {X 0,Y 191.006,Z 739.857,A -85,B 0,C 180,E1 -29724.22,E2 -29724.22} C_VEL
LIN {X 0,Y 192.19,Z 703.063,A -85,B 0,C 180,E1 -29726.735,E2 -29726.735} C_VEL
LIN {X 0,Y 193.144,Z 667.223,A -85,B 0,C 180,E1 -29729.049,E2 -29729.049} C_VEL
LIN {X 0,Y 190.7,Z 639.293,A -85,B 0,C 180,E1 -29730.785,E2 -29730.785} C_VEL
LIN {X 0,Y 190.47,Z 633.697,A -85,B 0,C 180,E1 -29731.204,E2 -29731.204} C_VEL
LIN {X 0,Y 189.705,Z 633.784,A -85,B 0,C 180,E1 -29738.878,E2 -29738.878} C_VEL
LIN {X 0,Y 189.701,Z 633.786,A -85,B 0,C 180,E1 -29742.398,E2 -29742.398} C_VEL
LIN {X 0,Y 189.701,Z 633.782,A -85,B 0,C 180,E1 -29747.6,E2 -29747.6} C_VEL
LIN {X 0,Y 189.693,Z 633.787,A -85,B 0,C 180,E1 -29751.117,E2 -29751.117} C_VEL
LIN {X 0,Y 189.65,Z 633.788,A -85,B 0,C 180,E1 -29756.357,E2 -29756.357} C_VEL
LIN {X 0,Y 189.706,Z 633.784,A -85,B 0,C 180,E1 -29758.874,E2 -29758.874} C_VEL
LIN {X 0,Y 189.729,Z 633.783,A -85,B 0,C 180,E1 -29763.703,E2 -29763.703} C_VEL
LIN {X 0,Y 189.795,Z 633.775,A -85,B 0,C 180,E1 -29768.342,E2 -29768.342} C_VEL
LIN {X 0,Y 189.923,Z 633.757,A -85,B 0,C 180,E1 -29773.511,E2 -29773.511} C_VEL
LIN {X 0,Y 189.962,Z 633.75,A -85,B 0,C 180,E1 -29777.218,E2 -29777.218} C_VEL
LIN {X 0,Y 190.388,Z 633.699,A -85,B 0,C 180,E1 -29783.663,E2 -29783.663} C_VEL
LIN {X 0,Y 190.49,Z 633.688,A -85,B 0,C 180,E1 -29787.892,E2 -29787.892} C_VEL
LIN {X 0,Y 190.575,Z 633.68,A -85,B 0,C 180,E1 -29790,E2 -29790} C_VEL
LIN {X 0,Y 190.411,Z 633.692,A -85,B 0,C 180,E1 -29794.219,E2 -29794.219} C_VEL
LIN {X 0,Y 190.369,Z 633.701,A -85,B 0,C 180,E1 -29796.575,E2 -29796.575} C_VEL
LIN {X 0,Y 189.961,Z 633.75,A -85,B 0,C 180,E1 -29802.781,E2 -29802.781} C_VEL
LIN {X 0,Y 189.859,Z 633.764,A -85,B 0,C 180,E1 -29807.166,E2 -29807.166} C_VEL
LIN {X 0,Y 189.795,Z 633.77,A -85,B 0,C 180,E1 -29812.689,E2 -29812.689} C_VEL
LIN {X 0,Y 189.734,Z 633.782,A -85,B 0,C 180,E1 -29817.626,E2 -29817.626} C_VEL
LIN {X 0,Y 189.716,Z 633.784,A -85,B 0,C 180,E1 -29821.88,E2 -29821.88} C_VEL
LIN {X 0,Y 189.687,Z 633.788,A -85,B 0,C 180,E1 -29826.215,E2 -29826.215} C_VEL
LIN {X 0,Y 189.689,Z 633.788,A -85,B 0,C 180,E1 -29829.156,E2 -29829.156} C_VEL
LIN {X 0,Y 189.701,Z 633.782,A -85,B 0,C 180,E1 -29832.4,E2 -29832.4} C_VEL
LIN {X 0,Y 189.701,Z 633.786,A -85,B 0,C 180,E1 -29837.601,E2 -29837.601} C_VEL
LIN {X 0,Y 189.707,Z 633.784,A -85,B 0,C 180,E1 -29841.122,E2 -29841.122} C_VEL
LIN {X 0,Y 189.671,Z 633.791,A -85,B 0,C 180,E1 -29846.363,E2 -29846.363} C_VEL
LIN {X 0,Y 189.707,Z 633.785,A -85,B 0,C 180,E1 -29848.876,E2 -29848.876} C_VEL
LIN {X 0,Y 189.734,Z 633.776,A -85,B 0,C 180,E1 -29853.705,E2 -29853.705} C_VEL
LIN {X 0,Y 189.747,Z 633.782,A -85,B 0,C 180,E1 -29858.338,E2 -29858.338} C_VEL
LIN {X 0,Y 189.875,Z 633.758,A -85,B 0,C 180,E1 -29863.562,E2 -29863.562} C_VEL
LIN {X 0,Y 189.998,Z 633.749,A -85,B 0,C 180,E1 -29869.379,E2 -29869.379} C_VEL
LIN {X 0,Y 190.39,Z 633.695,A -85,B 0,C 180,E1 -29873.664,E2 -29873.664} C_VEL
LIN {X 0,Y 190.496,Z 633.69,A -85,B 0,C 180,E1 -29877.893,E2 -29877.893} C_VEL
LIN {X 0,Y 190.575,Z 633.677,A -85,B 0,C 180,E1 -29880.001,E2 -29880.001} C_VEL
LIN {X 0,Y 190.414,Z 633.696,A -85,B 0,C 180,E1 -29884.22,E2 -29884.22} C_VEL
LIN {X 0,Y 190.371,Z 633.703,A -85,B 0,C 180,E1 -29886.576,E2 -29886.576} C_VEL
LIN {X 0,Y 189.898,Z 633.756,A -85,B 0,C 180,E1 -29892.787,E2 -29892.787} C_VEL
LIN {X 0,Y 189.783,Z 633.776,A -85,B 0,C 180,E1 -29897.174,E2 -29897.174} C_VEL
LIN {X 0,Y 189.763,Z 633.774,A -85,B 0,C 180,E1 -29902.664,E2 -29902.664} C_VEL
LIN {X 0,Y 189.736,Z 633.783,A -85,B 0,C 180,E1 -29907.626,E2 -29907.626} C_VEL
LIN {X 0,Y 189.693,Z 633.782,A -85,B 0,C 180,E1 -29911.867,E2 -29911.867} C_VEL
LIN {X 0,Y 189.656,Z 633.794,A -85,B 0,C 180,E1 -29916.223,E2 -29916.223} C_VEL
LIN {X 0,Y 189.66,Z 633.789,A -85,B 0,C 180,E1 -29919.144,E2 -29919.144} C_VEL
LIN {X 0,Y 189.635,Z 633.792,A -85,B 0,C 180,E1 -29922.377,E2 -29922.377} C_VEL
LIN {X 0,Y 189.635,Z 633.795,A -85,B 0,C 180,E1 -29927.624,E2 -29927.624} C_VEL
LIN {X 0,Y 189.681,Z 633.781,A -85,B 0,C 180,E1 -29931.115,E2 -29931.115} C_VEL
LIN {X 0,Y 189.652,Z 633.793,A -85,B 0,C 180,E1 -29936.359,E2 -29936.359} C_VEL
LIN {X 0,Y 189.833,Z 633.763,A -85,B 0,C 180,E1 -29941.336,E2 -29941.336} C_VEL
LIN {X 0,Y 190.56,Z 633.811,A -85,B 0,C 180,E1 -29945.43,E2 -29945.43} C_VEL
LIN {X 0,Y 190.778,Z 635.306,A -85,B 0,C 180,E1 -29946.18,E2 -29946.18} C_VEL
LIN {X 0,Y 189.917,Z 640.325,A -85,B 0,C 180,E1 -29948.713,E2 -29948.713} C_VEL
LIN {X 0,Y 190.6,Z 663.153,A -85,B 0,C 180,E1 -29950.163,E2 -29950.163} C_VEL
LIN {X 0,Y 192.819,Z 691.205,A -85,B 0,C 180,E1 -29951.911,E2 -29951.911} C_VEL
LIN {X 0,Y 191.464,Z 745.292,A -85,B 0,C 180,E1 -29955.501,E2 -29955.501} C_VEL
LIN {X 0,Y 191.081,Z 756.607,A -85,B 0,C 180,E1 -29956.486,E2 -29956.486} C_VEL
LIN {X 0,Y 190.706,Z 767.091,A -85,B 0,C 180,E1 -29957.674,E2 -29957.674} C_VEL
LIN {X 0,Y 190.329,Z 777.382,A -85,B 0,C 180,E1 -29959.129,E2 -29959.129} C_VEL
LIN {X 0,Y 189.872,Z 786.572,A -85,B 0,C 180,E1 -29960.713,E2 -29960.713} C_VEL
LIN {X 0,Y 189.48,Z 796.769,A -85,B 0,C 180,E1 -29962.833,E2 -29962.833} C_VEL
LIN {X 0,Y 189.262,Z 804.339,A -85,B 0,C 180,E1 -29964.692,E2 -29964.692} C_VEL
LIN {X 0,Y 189.129,Z 811.766,A -85,B 0,C 180,E1 -29966.816,E2 -29966.816} C_VEL
LIN {X 0,Y 189.032,Z 819.51,A -85,B 0,C 180,E1 -29969.47,E2 -29969.47} C_VEL
LIN {X 0,Y 188.858,Z 825.811,A -85,B 0,C 180,E1 -29972.126,E2 -29972.126} C_VEL
LIN {X 0,Y 188.371,Z 831.854,A -85,B 0,C 180,E1 -29975.334,E2 -29975.334} C_VEL
LIN {X 0,Y 188.18,Z 836.766,A -85,B 0,C 180,E1 -29978.563,E2 -29978.563} C_VEL
LIN {X 0,Y 188.785,Z 840.736,A -85,B 0,C 180,E1 -29981.775,E2 -29981.775} C_VEL
LIN {X 0,Y 190.221,Z 843.775,A -85,B 0,C 180,E1 -29984.938,E2 -29984.938} C_VEL
LIN {X 0,Y 193.3,Z 846.707,A -85,B 0,C 180,E1 -29989.034,E2 -29989.034} C_VEL
LIN {X 0,Y 197.638,Z 848.194,A -85,B 0,C 180,E1 -29992.946,E2 -29992.946} C_VEL
LIN {X 0,Y 203.168,Z 848.313,A -85,B 0,C 180,E1 -29996.628,E2 -29996.628} C_VEL
LIN {X 0,Y 206.286,Z 847.894,A -85,B 0,C 180,E1 -29998.384,E2 -29998.384} C_VEL
LIN {X 0,Y 213.469,Z 846.026,A -85,B 0,C 180,E1 -30001.669,E2 -30001.669} C_VEL
LIN {X 0,Y 221.534,Z 842.643,A -85,B 0,C 180,E1 -30004.689,E2 -30004.689} C_VEL
LIN {X 0,Y 222.885,Z 841.907,A -85,B 0,C 180,E1 -30005.149,E2 -30005.149} C_VEL
LIN {X 0,Y 225.853,Z 840.167,A -85,B 0,C 180,E1 -30006.375,E2 -30006.375} C_VEL
LIN {X 0,Y 233.323,Z 834.263,A -85,B 0,C 180,E1 -30010.415,E2 -30010.415} C_VEL
LIN {X 0,Y 235.939,Z 832.17,A -85,B 0,C 180,E1 -30011.293,E2 -30011.293} C_VEL
LIN {X 0,Y 237.157,Z 831.26,A -85,B 0,C 180,E1 -30011.594,E2 -30011.594} C_VEL
LIN {X 0,Y 245.211,Z 824.944,A -85,B 0,C 180,E1 -30013.28,E2 -30013.28} C_VEL
LIN {X 0,Y 252.115,Z 818.749,A -85,B 0,C 180,E1 -30014.549,E2 -30014.549} C_VEL
LIN {X 0,Y 257.775,Z 813.048,A -85,B 0,C 180,E1 -30015.503,E2 -30015.503} C_VEL
LIN {X 0,Y 265.217,Z 804.427,A -85,B 0,C 180,E1 -30016.633,E2 -30016.633} C_VEL
LIN {X 0,Y 271.814,Z 795.726,A -85,B 0,C 180,E1 -30017.532,E2 -30017.532} C_VEL
LIN {X 0,Y 277.942,Z 786.422,A -85,B 0,C 180,E1 -30018.296,E2 -30018.296} C_VEL
LIN {X 0,Y 283.246,Z 777.042,A -85,B 0,C 180,E1 -30018.918,E2 -30018.918} C_VEL
LIN {X 0,Y 288.139,Z 766.817,A -85,B 0,C 180,E1 -30019.449,E2 -30019.449} C_VEL
LIN {X 0,Y 288.235,Z 766.349,A -85,B 0,C 180,E1 -30019.983,E2 -30019.983} C_VEL
LIN {X 0,Y 288.331,Z 766.151,A -85,B 0,C 180,E1 -30020.83,E2 -30020.83} C_VEL
LIN {X 0,Y 287.729,Z 767.611,A -85,B 0,C 180,E1 -30021.035,E2 -30021.035} C_VEL
LIN {X 0,Y 280.817,Z 781.205,A -85,B 0,C 180,E1 -30021.877,E2 -30021.877} C_VEL
LIN {X 0,Y 274.199,Z 791.739,A -85,B 0,C 180,E1 -30022.784,E2 -30022.784} C_VEL
LIN {X 0,Y 268.556,Z 799.492,A -85,B 0,C 180,E1 -30023.604,E2 -30023.604} C_VEL
LIN {X 0,Y 261.169,Z 808.394,A -85,B 0,C 180,E1 -30024.786,E2 -30024.786} C_VEL
LIN {X 0,Y 254.744,Z 815.126,A -85,B 0,C 180,E1 -30025.905,E2 -30025.905} C_VEL
LIN {X 0,Y 246.947,Z 822.136,A -85,B 0,C 180,E1 -30027.39,E2 -30027.39} C_VEL
LIN {X 0,Y 238.901,Z 828.333,A -85,B 0,C 180,E1 -30029.13,E2 -30029.13} C_VEL
LIN {X 0,Y 231.233,Z 833.342,A -85,B 0,C 180,E1 -30031.009,E2 -30031.009} C_VEL
LIN {X 0,Y 223.865,Z 837.277,A -85,B 0,C 180,E1 -30033.019,E2 -30033.019} C_VEL
LIN {X 0,Y 214.838,Z 840.948,A -85,B 0,C 180,E1 -30035.909,E2 -30035.909} C_VEL
LIN {X 0,Y 208.51,Z 842.706,A -85,B 0,C 180,E1 -30038.313,E2 -30038.313} C_VEL
LIN {X 0,Y 204.573,Z 843.48,A -85,B 0,C 180,E1 -30039.977,E2 -30039.977} C_VEL
LIN {X 0,Y 196.908,Z 843.593,A -85,B 0,C 180,E1 -30043.833,E2 -30043.833} C_VEL
LIN {X 0,Y 191.66,Z 842.422,A -85,B 0,C 180,E1 -30047.333,E2 -30047.333} C_VEL
LIN {X 0,Y 189.094,Z 841.367,A -85,B 0,C 180,E1 -30049.326,E2 -30049.326} C_VEL
LIN {X 0,Y 185.097,Z 838.014,A -85,B 0,C 180,E1 -30053.481,E2 -30053.481} C_VEL
LIN {X 0,Y 183.026,Z 834.557,A -85,B 0,C 180,E1 -30056.708,E2 -30056.708} C_VEL
LIN {X 0,Y 181.271,Z 828.446,A -85,B 0,C 180,E1 -30061.106,E2 -30061.106} C_VEL
LIN {X 0,Y 180.698,Z 822.744,A -85,B 0,C 180,E1 -30064.446,E2 -30064.446} C_VEL
LIN {X 0,Y 180.795,Z 815.757,A -85,B 0,C 180,E1 -30067.792,E2 -30067.792} C_VEL
LIN {X 0,Y 181.058,Z 808.735,A -85,B 0,C 180,E1 -30070.588,E2 -30070.588} C_VEL
LIN {X 0,Y 181.471,Z 800.277,A -85,B 0,C 180,E1 -30073.39,E2 -30073.39} C_VEL
LIN {X 0,Y 181.761,Z 790.921,A -85,B 0,C 180,E1 -30075.936,E2 -30075.936} C_VEL
LIN {X 0,Y 182.159,Z 782.29,A -85,B 0,C 180,E1 -30077.915,E2 -30077.915} C_VEL
LIN {X 0,Y 182.627,Z 771.733,A -85,B 0,C 180,E1 -30079.9,E2 -30079.9} C_VEL
LIN {X 0,Y 183.21,Z 760.713,A -85,B 0,C 180,E1 -30081.59,E2 -30081.59} C_VEL
LIN {X 0,Y 183.695,Z 750.179,A -85,B 0,C 180,E1 -30082.881,E2 -30082.881} C_VEL
LIN {X 0,Y 184.033,Z 738.885,A -85,B 0,C 180,E1 -30083.946,E2 -30083.946} C_VEL
LIN {X 0,Y 185.369,Z 693.801,A -85,B 0,C 180,E1 -30087.115,E2 -30087.115} C_VEL
LIN {X 0,Y 186.105,Z 667.773,A -85,B 0,C 180,E1 -30088.879,E2 -30088.879} C_VEL
LIN {X 0,Y 183.643,Z 639.86,A -85,B 0,C 180,E1 -30090.698,E2 -30090.698} C_VEL
LIN {X 0,Y 183.395,Z 634.579,A -85,B 0,C 180,E1 -30091.116,E2 -30091.116} C_VEL
LIN {X 0,Y 182.636,Z 634.662,A -85,B 0,C 180,E1 -30097.851,E2 -30097.851} C_VEL
LIN {X 0,Y 182.64,Z 634.665,A -85,B 0,C 180,E1 -30103.224,E2 -30103.224} C_VEL
LIN {X 0,Y 182.64,Z 634.66,A -85,B 0,C 180,E1 -30106.774,E2 -30106.774} C_VEL
LIN {X 0,Y 182.591,Z 634.673,A -85,B 0,C 180,E1 -30112.136,E2 -30112.136} C_VEL
LIN {X 0,Y 182.613,Z 634.665,A -85,B 0,C 180,E1 -30117.547,E2 -30117.547} C_VEL
LIN {X 0,Y 182.692,Z 634.658,A -85,B 0,C 180,E1 -30122.607,E2 -30122.607} C_VEL
LIN {X 0,Y 182.772,Z 634.646,A -85,B 0,C 180,E1 -30127.465,E2 -30127.465} C_VEL
LIN {X 0,Y 182.871,Z 634.635,A -85,B 0,C 180,E1 -30133.245,E2 -30133.245} C_VEL
LIN {X 0,Y 182.96,Z 634.625,A -85,B 0,C 180,E1 -30138.964,E2 -30138.964} C_VEL
LIN {X 0,Y 183.321,Z 634.579,A -85,B 0,C 180,E1 -30143.418,E2 -30143.418} C_VEL
LIN {X 0,Y 183.457,Z 634.563,A -85,B 0,C 180,E1 -30147.811,E2 -30147.811} C_VEL
LIN {X 0,Y 183.539,Z 634.557,A -85,B 0,C 180,E1 -30150,E2 -30150} C_VEL
LIN {X 0,Y 183.354,Z 634.57,A -85,B 0,C 180,E1 -30154.381,E2 -30154.381} C_VEL
LIN {X 0,Y 183.32,Z 634.579,A -85,B 0,C 180,E1 -30156.582,E2 -30156.582} C_VEL
LIN {X 0,Y 182.96,Z 634.625,A -85,B 0,C 180,E1 -30161.035,E2 -30161.035} C_VEL
LIN {X 0,Y 182.87,Z 634.635,A -85,B 0,C 180,E1 -30166.754,E2 -30166.754} C_VEL
LIN {X 0,Y 182.771,Z 634.646,A -85,B 0,C 180,E1 -30172.534,E2 -30172.534} C_VEL
LIN {X 0,Y 182.682,Z 634.663,A -85,B 0,C 180,E1 -30178.133,E2 -30178.133} C_VEL
LIN {X 0,Y 182.65,Z 634.66,A -85,B 0,C 180,E1 -30182.471,E2 -30182.471} C_VEL
LIN {X 0,Y 182.612,Z 634.67,A -85,B 0,C 180,E1 -30187.858,E2 -30187.858} C_VEL
LIN {X 0,Y 182.64,Z 634.66,A -85,B 0,C 180,E1 -30193.226,E2 -30193.226} C_VEL
LIN {X 0,Y 182.64,Z 634.665,A -85,B 0,C 180,E1 -30196.775,E2 -30196.775} C_VEL
LIN {X 0,Y 182.604,Z 634.666,A -85,B 0,C 180,E1 -30202.141,E2 -30202.141} C_VEL
LIN {X 0,Y 182.634,Z 634.667,A -85,B 0,C 180,E1 -30207.538,E2 -30207.538} C_VEL
LIN {X 0,Y 182.698,Z 634.651,A -85,B 0,C 180,E1 -30212.61,E2 -30212.61} C_VEL
LIN {X 0,Y 182.74,Z 634.654,A -85,B 0,C 180,E1 -30217.463,E2 -30217.463} C_VEL
LIN {X 0,Y 182.834,Z 634.634,A -85,B 0,C 180,E1 -30223.286,E2 -30223.286} C_VEL
LIN {X 0,Y 182.939,Z 634.628,A -85,B 0,C 180,E1 -30228.964,E2 -30228.964} C_VEL
LIN {X 0,Y 183.322,Z 634.574,A -85,B 0,C 180,E1 -30233.419,E2 -30233.419} C_VEL
LIN {X 0,Y 183.463,Z 634.565,A -85,B 0,C 180,E1 -30237.813,E2 -30237.813} C_VEL
LIN {X 0,Y 183.539,Z 634.553,A -85,B 0,C 180,E1 -30240.001,E2 -30240.001} C_VEL
LIN {X 0,Y 183.357,Z 634.576,A -85,B 0,C 180,E1 -30244.382,E2 -30244.382} C_VEL
LIN {X 0,Y 183.323,Z 634.581,A -85,B 0,C 180,E1 -30246.583,E2 -30246.583} C_VEL
LIN {X 0,Y 182.935,Z 634.624,A -85,B 0,C 180,E1 -30251.038,E2 -30251.038} C_VEL
LIN {X 0,Y 182.77,Z 634.65,A -85,B 0,C 180,E1 -30256.647,E2 -30256.647} C_VEL
LIN {X 0,Y 182.739,Z 634.649,A -85,B 0,C 180,E1 -30262.539,E2 -30262.539} C_VEL
LIN {X 0,Y 182.681,Z 634.661,A -85,B 0,C 180,E1 -30268.131,E2 -30268.131} C_VEL
LIN {X 0,Y 182.613,Z 634.666,A -85,B 0,C 180,E1 -30272.48,E2 -30272.48} C_VEL
LIN {X 0,Y 182.587,Z 634.675,A -85,B 0,C 180,E1 -30277.865,E2 -30277.865} C_VEL
LIN {X 0,Y 182.587,Z 634.665,A -85,B 0,C 180,E1 -30280.705,E2 -30280.705} C_VEL
LIN {X 0,Y 182.554,Z 634.674,A -85,B 0,C 180,E1 -30283.682,E2 -30283.682} C_VEL
LIN {X 0,Y 182.56,Z 634.676,A -85,B 0,C 180,E1 -30286.802,E2 -30286.802} C_VEL
LIN {X 0,Y 182.595,Z 634.666,A -85,B 0,C 180,E1 -30290.105,E2 -30290.105} C_VEL
LIN {X 0,Y 182.589,Z 634.672,A -85,B 0,C 180,E1 -30294.871,E2 -30294.871} C_VEL
LIN {X 0,Y 182.698,Z 634.653,A -85,B 0,C 180,E1 -30300.106,E2 -30300.106} C_VEL
LIN {X 0,Y 183.602,Z 634.663,A -85,B 0,C 180,E1 -30305.871,E2 -30305.871} C_VEL
LIN {X 0,Y 182.83,Z 640.12,A -85,B 0,C 180,E1 -30308.731,E2 -30308.731} C_VEL
LIN {X 0,Y 183.533,Z 663.513,A -85,B 0,C 180,E1 -30310.305,E2 -30310.305} C_VEL
LIN {X 0,Y 185.736,Z 692.266,A -85,B 0,C 180,E1 -30312.182,E2 -30312.182} C_VEL
LIN {X 0,Y 184.456,Z 744.971,A -85,B 0,C 180,E1 -30315.851,E2 -30315.851} C_VEL
LIN {X 0,Y 184.11,Z 756.977,A -85,B 0,C 180,E1 -30316.945,E2 -30316.945} C_VEL
LIN {X 0,Y 183.724,Z 768.336,A -85,B 0,C 180,E1 -30318.315,E2 -30318.315} C_VEL
LIN {X 0,Y 183.31,Z 778.287,A -85,B 0,C 180,E1 -30319.821,E2 -30319.821} C_VEL
LIN {X 0,Y 182.915,Z 787.294,A -85,B 0,C 180,E1 -30321.467,E2 -30321.467} C_VEL
LIN {X 0,Y 182.608,Z 796.184,A -85,B 0,C 180,E1 -30323.393,E2 -30323.393} C_VEL
LIN {X 0,Y 182.403,Z 804.74,A -85,B 0,C 180,E1 -30325.596,E2 -30325.596} C_VEL
LIN {X 0,Y 182.377,Z 811.972,A -85,B 0,C 180,E1 -30327.799,E2 -30327.799} C_VEL
LIN {X 0,Y 182.267,Z 819.474,A -85,B 0,C 180,E1 -30330.551,E2 -30330.551} C_VEL
LIN {X 0,Y 181.976,Z 825.652,A -85,B 0,C 180,E1 -30333.31,E2 -30333.31} C_VEL
LIN {X 0,Y 181.482,Z 831.624,A -85,B 0,C 180,E1 -30336.649,E2 -30336.649} C_VEL
LIN {X 0,Y 181.487,Z 836.462,A -85,B 0,C 180,E1 -30340.002,E2 -30340.002} C_VEL
LIN {X 0,Y 182.939,Z 841.451,A -85,B 0,C 180,E1 -30344.411,E2 -30344.411} C_VEL
LIN {X 0,Y 184.831,Z 844.328,A -85,B 0,C 180,E1 -30347.649,E2 -30347.649} C_VEL
LIN {X 0,Y 188.703,Z 846.838,A -85,B 0,C 180,E1 -30351.789,E2 -30351.789} C_VEL
LIN {X 0,Y 193.818,Z 848.034,A -85,B 0,C 180,E1 -30355.701,E2 -30355.701} C_VEL
LIN {X 0,Y 196.868,Z 848.224,A -85,B 0,C 180,E1 -30357.551,E2 -30357.551} C_VEL
LIN {X 0,Y 203.657,Z 847.438,A -85,B 0,C 180,E1 -30361.058,E2 -30361.058} C_VEL
LIN {X 0,Y 211.537,Z 845.209,A -85,B 0,C 180,E1 -30364.257,E2 -30364.257} C_VEL
LIN {X 0,Y 217.963,Z 842.645,A -85,B 0,C 180,E1 -30366.479,E2 -30366.479} C_VEL
LIN {X 0,Y 227.248,Z 837.79,A -85,B 0,C 180,E1 -30369.189,E2 -30369.189} C_VEL
LIN {X 0,Y 234.702,Z 833.05,A -85,B 0,C 180,E1 -30371.039,E2 -30371.039} C_VEL
LIN {X 0,Y 237.157,Z 831.26,A -85,B 0,C 180,E1 -30371.594,E2 -30371.594} C_VEL
LIN {X 0,Y 240.611,Z 828.617,A -85,B 0,C 180,E1 -30372.544,E2 -30372.544} C_VEL
LIN {X 0,Y 249.619,Z 819.985,A -85,B 0,C 180,E1 -30375.826,E2 -30375.826} C_VEL
LIN {X 0,Y 252.432,Z 817.187,A -85,B 0,C 180,E1 -30376.495,E2 -30376.495} C_VEL
LIN {X 0,Y 253.689,Z 816.001,A -85,B 0,C 180,E1 -30376.711,E2 -30376.711} C_VEL
LIN {X 0,Y 263.486,Z 805.656,A -85,B 0,C 180,E1 -30378.103,E2 -30378.103} C_VEL
LIN {X 0,Y 271.145,Z 795.91,A -85,B 0,C 180,E1 -30379.079,E2 -30379.079} C_VEL
LIN {X 0,Y 277.419,Z 786.601,A -85,B 0,C 180,E1 -30379.798,E2 -30379.798} C_VEL
LIN {X 0,Y 280.253,Z 781.889,A -85,B 0,C 180,E1 -30380.104,E2 -30380.104} C_VEL
LIN {X 0,Y 280.286,Z 781.79,A -85,B 0,C 180,E1 -30380.412,E2 -30380.412} C_VEL
LIN {X 0,Y 273.946,Z 791.721,A -85,B 0,C 180,E1 -30381.212,E2 -30381.212} C_VEL
LIN {X 0,Y 267.438,Z 800.425,A -85,B 0,C 180,E1 -30382.092,E2 -30382.092} C_VEL
LIN {X 0,Y 261.547,Z 807.329,A -85,B 0,C 180,E1 -30382.946,E2 -30382.946} C_VEL
LIN {X 0,Y 254.052,Z 814.927,A -85,B 0,C 180,E1 -30384.134,E2 -30384.134} C_VEL
LIN {X 0,Y 246.753,Z 821.456,A -85,B 0,C 180,E1 -30385.408,E2 -30385.408} C_VEL
LIN {X 0,Y 238.283,Z 827.847,A -85,B 0,C 180,E1 -30387.056,E2 -30387.056} C_VEL
LIN {X 0,Y 230.228,Z 832.938,A -85,B 0,C 180,E1 -30388.854,E2 -30388.854} C_VEL
LIN {X 0,Y 222.468,Z 837.051,A -85,B 0,C 180,E1 -30390.789,E2 -30390.789} C_VEL
LIN {X 0,Y 215.114,Z 840.152,A -85,B 0,C 180,E1 -30392.879,E2 -30392.879} C_VEL
LIN {X 0,Y 208.798,Z 842.155,A -85,B 0,C 180,E1 -30394.926,E2 -30394.926} C_VEL
LIN {X 0,Y 201.815,Z 843.583,A -85,B 0,C 180,E1 -30397.555,E2 -30397.555} C_VEL
LIN {X 0,Y 194.049,Z 843.997,A -85,B 0,C 180,E1 -30401.042,E2 -30401.042} C_VEL
LIN {X 0,Y 187.51,Z 842.92,A -85,B 0,C 180,E1 -30404.841,E2 -30404.841} C_VEL
LIN {X 0,Y 184.661,Z 841.874,A -85,B 0,C 180,E1 -30406.844,E2 -30406.844} C_VEL
LIN {X 0,Y 179.879,Z 838.76,A -85,B 0,C 180,E1 -30411.039,E2 -30411.039} C_VEL
LIN {X 0,Y 176.646,Z 834.182,A -85,B 0,C 180,E1 -30415.451,E2 -30415.451} C_VEL
LIN {X 0,Y 174.906,Z 829.066,A -85,B 0,C 180,E1 -30419.267,E2 -30419.267} C_VEL
LIN {X 0,Y 174.052,Z 823.195,A -85,B 0,C 180,E1 -30422.883,E2 -30422.883} C_VEL
LIN {X 0,Y 173.926,Z 816.448,A -85,B 0,C 180,E1 -30426.358,E2 -30426.358} C_VEL
LIN {X 0,Y 174.173,Z 809.661,A -85,B 0,C 180,E1 -30429.256,E2 -30429.256} C_VEL
LIN {X 0,Y 174.519,Z 801.41,A -85,B 0,C 180,E1 -30432.163,E2 -30432.163} C_VEL
LIN {X 0,Y 174.812,Z 791.885,A -85,B 0,C 180,E1 -30434.915,E2 -30434.915} C_VEL
LIN {X 0,Y 175.222,Z 782.674,A -85,B 0,C 180,E1 -30437.146,E2 -30437.146} C_VEL
LIN {X 0,Y 175.683,Z 772.431,A -85,B 0,C 180,E1 -30439.203,E2 -30439.203} C_VEL
LIN {X 0,Y 176.19,Z 761.711,A -85,B 0,C 180,E1 -30440.964,E2 -30440.964} C_VEL
LIN {X 0,Y 176.632,Z 751.76,A -85,B 0,C 180,E1 -30442.284,E2 -30442.284} C_VEL
LIN {X 0,Y 176.972,Z 740.988,A -85,B 0,C 180,E1 -30443.389,E2 -30443.389} C_VEL
LIN {X 0,Y 177.964,Z 706.563,A -85,B 0,C 180,E1 -30445.967,E2 -30445.967} C_VEL
LIN {X 0,Y 179.014,Z 667.853,A -85,B 0,C 180,E1 -30448.708,E2 -30448.708} C_VEL
LIN {X 0,Y 176.57,Z 640.08,A -85,B 0,C 180,E1 -30450.591,E2 -30450.591} C_VEL
LIN {X 0,Y 176.357,Z 635.456,A -85,B 0,C 180,E1 -30450.984,E2 -30450.984} C_VEL
LIN {X 0,Y 175.613,Z 635.534,A -85,B 0,C 180,E1 -30457.087,E2 -30457.087} C_VEL
LIN {X 0,Y 175.579,Z 635.545,A -85,B 0,C 180,E1 -30462.701,E2 -30462.701} C_VEL
LIN {X 0,Y 175.578,Z 635.54,A -85,B 0,C 180,E1 -30467.297,E2 -30467.297} C_VEL
LIN {X 0,Y 175.551,Z 635.55,A -85,B 0,C 180,E1 -30470.327,E2 -30470.327} C_VEL
LIN {X 0,Y 175.574,Z 635.545,A -85,B 0,C 180,E1 -30473.243,E2 -30473.243} C_VEL
LIN {X 0,Y 175.552,Z 635.548,A -85,B 0,C 180,E1 -30478.755,E2 -30478.755} C_VEL
LIN {X 0,Y 175.606,Z 635.542,A -85,B 0,C 180,E1 -30481.402,E2 -30481.402} C_VEL
LIN {X 0,Y 175.668,Z 635.531,A -85,B 0,C 180,E1 -30486.501,E2 -30486.501} C_VEL
LIN {X 0,Y 175.702,Z 635.531,A -85,B 0,C 180,E1 -30491.402,E2 -30491.402} C_VEL
LIN {X 0,Y 175.83,Z 635.512,A -85,B 0,C 180,E1 -30493.808,E2 -30493.808} C_VEL
LIN {X 0,Y 175.882,Z 635.508,A -85,B 0,C 180,E1 -30498.514,E2 -30498.514} C_VEL
LIN {X 0,Y 176.266,Z 635.458,A -85,B 0,C 180,E1 -30503.427,E2 -30503.427} C_VEL
LIN {X 0,Y 176.424,Z 635.439,A -85,B 0,C 180,E1 -30507.724,E2 -30507.724} C_VEL
LIN {X 0,Y 176.504,Z 635.433,A -85,B 0,C 180,E1 -30510,E2 -30510} C_VEL
LIN {X 0,Y 176.295,Z 635.449,A -85,B 0,C 180,E1 -30514.557,E2 -30514.557} C_VEL
LIN {X 0,Y 176.228,Z 635.462,A -85,B 0,C 180,E1 -30516.848,E2 -30516.848} C_VEL
LIN {X 0,Y 175.881,Z 635.508,A -85,B 0,C 180,E1 -30521.485,E2 -30521.485} C_VEL
LIN {X 0,Y 175.801,Z 635.515,A -85,B 0,C 180,E1 -30527.018,E2 -30527.018} C_VEL
LIN {X 0,Y 175.663,Z 635.534,A -85,B 0,C 180,E1 -30531.03,E2 -30531.03} C_VEL
LIN {X 0,Y 175.667,Z 635.531,A -85,B 0,C 180,E1 -30533.499,E2 -30533.499} C_VEL
LIN {X 0,Y 175.612,Z 635.542,A -85,B 0,C 180,E1 -30538.661,E2 -30538.661} C_VEL
LIN {X 0,Y 175.544,Z 635.544,A -85,B 0,C 180,E1 -30543.96,E2 -30543.96} C_VEL
LIN {X 0,Y 175.592,Z 635.542,A -85,B 0,C 180,E1 -30547.08,E2 -30547.08} C_VEL
LIN {X 0,Y 175.579,Z 635.54,A -85,B 0,C 180,E1 -30552.702,E2 -30552.702} C_VEL
LIN {X 0,Y 175.579,Z 635.545,A -85,B 0,C 180,E1 -30557.299,E2 -30557.299} C_VEL
LIN {X 0,Y 175.559,Z 635.547,A -85,B 0,C 180,E1 -30560.331,E2 -30560.331} C_VEL
LIN {X 0,Y 175.588,Z 635.538,A -85,B 0,C 180,E1 -30563.248,E2 -30563.248} C_VEL
LIN {X 0,Y 175.562,Z 635.547,A -85,B 0,C 180,E1 -30568.758,E2 -30568.758} C_VEL
LIN {X 0,Y 175.624,Z 635.538,A -85,B 0,C 180,E1 -30571.407,E2 -30571.407} C_VEL
LIN {X 0,Y 175.633,Z 635.539,A -85,B 0,C 180,E1 -30576.529,E2 -30576.529} C_VEL
LIN {X 0,Y 175.687,Z 635.529,A -85,B 0,C 180,E1 -30581.401,E2 -30581.401} C_VEL
LIN {X 0,Y 175.798,Z 635.512,A -85,B 0,C 180,E1 -30583.806,E2 -30583.806} C_VEL
LIN {X 0,Y 175.857,Z 635.511,A -85,B 0,C 180,E1 -30588.513,E2 -30588.513} C_VEL
LIN {X 0,Y 176.268,Z 635.453,A -85,B 0,C 180,E1 -30593.429,E2 -30593.429} C_VEL
LIN {X 0,Y 176.43,Z 635.441,A -85,B 0,C 180,E1 -30597.725,E2 -30597.725} C_VEL
LIN {X 0,Y 176.504,Z 635.429,A -85,B 0,C 180,E1 -30600.001,E2 -30600.001} C_VEL
LIN {X 0,Y 176.298,Z 635.454,A -85,B 0,C 180,E1 -30604.558,E2 -30604.558} C_VEL
LIN {X 0,Y 176.23,Z 635.464,A -85,B 0,C 180,E1 -30606.849,E2 -30606.849} C_VEL
LIN {X 0,Y 175.851,Z 635.507,A -85,B 0,C 180,E1 -30611.488,E2 -30611.488} C_VEL
LIN {X 0,Y 175.718,Z 635.528,A -85,B 0,C 180,E1 -30616.927,E2 -30616.927} C_VEL
LIN {X 0,Y 175.62,Z 635.534,A -85,B 0,C 180,E1 -30621.037,E2 -30621.037} C_VEL
LIN {X 0,Y 175.594,Z 635.546,A -85,B 0,C 180,E1 -30626.027,E2 -30626.027} C_VEL
LIN {X 0,Y 175.615,Z 635.539,A -85,B 0,C 180,E1 -30628.662,E2 -30628.662} C_VEL
LIN {X 0,Y 175.51,Z 635.553,A -85,B 0,C 180,E1 -30633.968,E2 -30633.968} C_VEL
LIN {X 0,Y 175.542,Z 635.55,A -85,B 0,C 180,E1 -30637.058,E2 -30637.058} C_VEL
LIN {X 0,Y 175.557,Z 635.541,A -85,B 0,C 180,E1 -30640.706,E2 -30640.706} C_VEL
LIN {X 0,Y 175.505,Z 635.557,A -85,B 0,C 180,E1 -30645.922,E2 -30645.922} C_VEL
LIN {X 0,Y 175.537,Z 635.544,A -85,B 0,C 180,E1 -30650.324,E2 -30650.324} C_VEL
LIN {X 0,Y 175.57,Z 635.544,A -85,B 0,C 180,E1 -30653.243,E2 -30653.243} C_VEL
LIN {X 0,Y 175.593,Z 635.54,A -85,B 0,C 180,E1 -30658.764,E2 -30658.764} C_VEL
LIN {X 0,Y 176.511,Z 635.434,A -85,B 0,C 180,E1 -30666.282,E2 -30666.282} C_VEL
LIN {X 0,Y 175.738,Z 640.037,A -85,B 0,C 180,E1 -30668.826,E2 -30668.826} C_VEL
LIN {X 0,Y 176.491,Z 664.193,A -85,B 0,C 180,E1 -30670.518,E2 -30670.518} C_VEL
LIN {X 0,Y 178.699,Z 691.84,A -85,B 0,C 180,E1 -30672.39,E2 -30672.39} C_VEL
LIN {X 0,Y 177.459,Z 744.658,A -85,B 0,C 180,E1 -30676.229,E2 -30676.229} C_VEL
LIN {X 0,Y 177.117,Z 757.291,A -85,B 0,C 180,E1 -30677.438,E2 -30677.438} C_VEL
LIN {X 0,Y 176.789,Z 767.521,A -85,B 0,C 180,E1 -30678.719,E2 -30678.719} C_VEL
LIN {X 0,Y 176.394,Z 777.563,A -85,B 0,C 180,E1 -30680.284,E2 -30680.284} C_VEL
LIN {X 0,Y 176.005,Z 787.882,A -85,B 0,C 180,E1 -30682.281,E2 -30682.281} C_VEL
LIN {X 0,Y 175.777,Z 796.522,A -85,B 0,C 180,E1 -30684.283,E2 -30684.283} C_VEL
LIN {X 0,Y 175.623,Z 804.868,A -85,B 0,C 180,E1 -30686.571,E2 -30686.571} C_VEL
LIN {X 0,Y 175.628,Z 812.011,A -85,B 0,C 180,E1 -30688.858,E2 -30688.858} C_VEL
LIN {X 0,Y 175.503,Z 819.307,A -85,B 0,C 180,E1 -30691.672,E2 -30691.672} C_VEL
LIN {X 0,Y 175.084,Z 825.463,A -85,B 0,C 180,E1 -30694.59,E2 -30694.59} C_VEL
LIN {X 0,Y 174.666,Z 831.275,A -85,B 0,C 180,E1 -30698.069,E2 -30698.069} C_VEL
LIN {X 0,Y 174.975,Z 836.086,A -85,B 0,C 180,E1 -30701.547,E2 -30701.547} C_VEL
LIN {X 0,Y 176.768,Z 841.113,A -85,B 0,C 180,E1 -30706.104,E2 -30706.104} C_VEL
LIN {X 0,Y 180.09,Z 844.673,A -85,B 0,C 180,E1 -30710.491,E2 -30710.491} C_VEL
LIN {X 0,Y 182.729,Z 846.298,A -85,B 0,C 180,E1 -30713.076,E2 -30713.076} C_VEL
LIN {X 0,Y 187.46,Z 847.665,A -85,B 0,C 180,E1 -30716.64,E2 -30716.64} C_VEL
LIN {X 0,Y 193.924,Z 847.922,A -85,B 0,C 180,E1 -30720.377,E2 -30720.377} C_VEL
LIN {X 0,Y 201.555,Z 846.826,A -85,B 0,C 180,E1 -30723.782,E2 -30723.782} C_VEL
LIN {X 0,Y 210.103,Z 844.362,A -85,B 0,C 180,E1 -30726.877,E2 -30726.877} C_VEL
LIN {X 0,Y 217.031,Z 841.613,A -85,B 0,C 180,E1 -30729.002,E2 -30729.002} C_VEL
LIN {X 0,Y 224.344,Z 837.972,A -85,B 0,C 180,E1 -30730.97,E2 -30730.97} C_VEL
LIN {X 0,Y 233.116,Z 832.68,A -85,B 0,C 180,E1 -30732.97,E2 -30732.97} C_VEL
LIN {X 0,Y 241.624,Z 826.567,A -85,B 0,C 180,E1 -30734.668,E2 -30734.668} C_VEL
LIN {X 0,Y 248.71,Z 820.684,A -85,B 0,C 180,E1 -30735.903,E2 -30735.903} C_VEL
LIN {X 0,Y 253.689,Z 816.001,A -85,B 0,C 180,E1 -30736.711,E2 -30736.711} C_VEL
LIN {X 0,Y 256.039,Z 813.729,A -85,B 0,C 180,E1 -30737.235,E2 -30737.235} C_VEL
LIN {X 0,Y 261.992,Z 806.883,A -85,B 0,C 180,E1 -30739.45,E2 -30739.45} C_VEL
LIN {X 0,Y 264.177,Z 804.216,A -85,B 0,C 180,E1 -30739.877,E2 -30739.877} C_VEL
LIN {X 0,Y 267.023,Z 800.769,A -85,B 0,C 180,E1 -30740.214,E2 -30740.214} C_VEL
LIN {X 0,Y 267.001,Z 800.772,A -85,B 0,C 180,E1 -30740.508,E2 -30740.508} C_VEL
LIN {X 0,Y 259.524,Z 809.161,A -85,B 0,C 180,E1 -30741.509,E2 -30741.509} C_VEL
LIN {X 0,Y 252.983,Z 815.545,A -85,B 0,C 180,E1 -30742.474,E2 -30742.474} C_VEL
LIN {X 0,Y 244.831,Z 822.374,A -85,B 0,C 180,E1 -30743.781,E2 -30743.781} C_VEL
LIN {X 0,Y 238.066,Z 827.376,A -85,B 0,C 180,E1 -30744.988,E2 -30744.988} C_VEL
LIN {X 0,Y 229.607,Z 832.674,A -85,B 0,C 180,E1 -30746.693,E2 -30746.693} C_VEL
LIN {X 0,Y 222.013,Z 836.614,A -85,B 0,C 180,E1 -30748.413,E2 -30748.413} C_VEL
LIN {X 0,Y 213.656,Z 840.059,A -85,B 0,C 180,E1 -30750.543,E2 -30750.543} C_VEL
LIN {X 0,Y 202.905,Z 843.021,A -85,B 0,C 180,E1 -30753.838,E2 -30753.838} C_VEL
LIN {X 0,Y 195.132,Z 844.077,A -85,B 0,C 180,E1 -30756.742,E2 -30756.742} C_VEL
